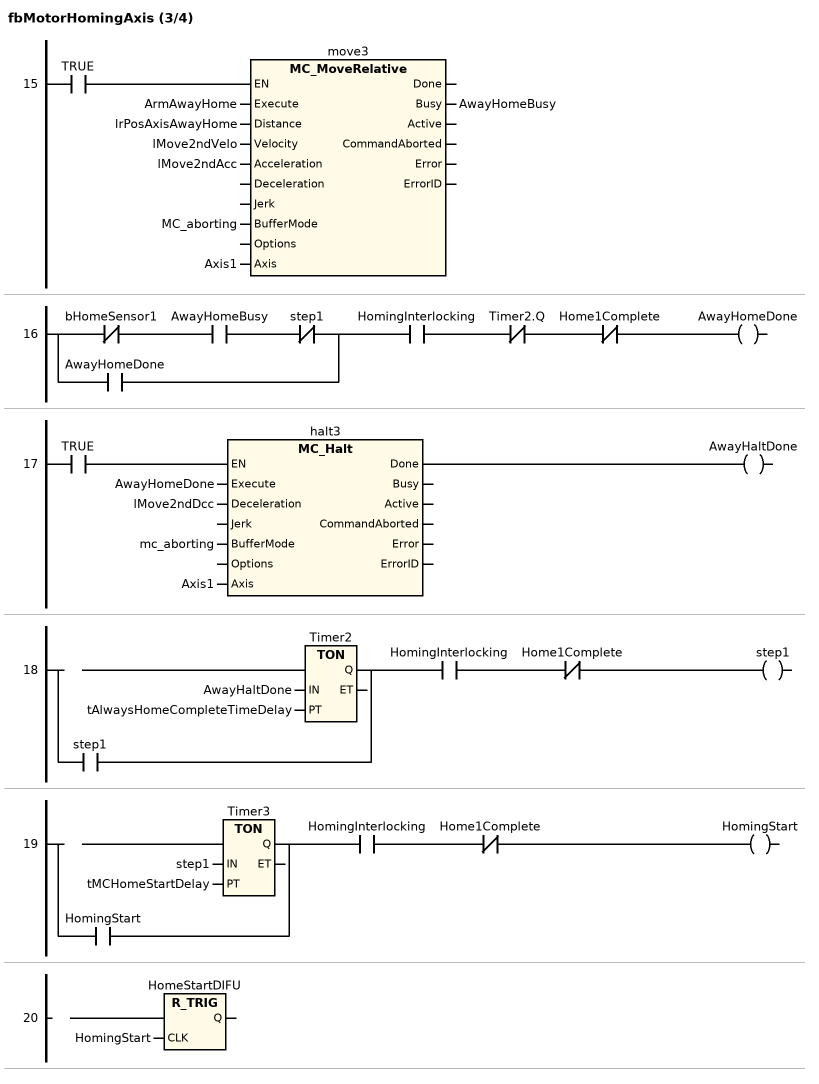
// NETWORK 15
move3(
    Execute := ArmAwayHome,
    Distance := lrPosAxisAwayHome,
    Velocity := lMove2ndVelo,
    Acceleration := lMove2ndAcc,
    BufferMode := MC_aborting,
    Axis := Axis1,
    Busy => AwayHomeBusy); // MC_MoveRelative

// NETWORK 16
AwayHomeDone := (NOT bHomeSensor1 AND AwayHomeBusy AND NOT step1 OR AwayHomeDone) AND HomingInterlocking AND NOT Timer2.Q AND NOT Home1Complete;

// NETWORK 17
halt3(Execute := AwayHomeDone, Deceleration := lMove2ndDcc, BufferMode := mc_aborting, Axis := Axis1); // MC_Halt
AwayHaltDone := halt3.Done;

// NETWORK 18
Timer2(IN := AwayHaltDone, PT := tAlwaysHomeCompleteTimeDelay); // TON
step1 := (Timer2.Q OR step1) AND HomingInterlocking AND NOT Home1Complete;

// NETWORK 19
Timer3(IN := step1, PT := tMCHomeStartDelay); // TON
HomingStart := (Timer3.Q OR HomingStart) AND HomingInterlocking AND NOT Home1Complete;

// NETWORK 20
HomeStartDIFU(CLK := HomingStart); // R_TRIG

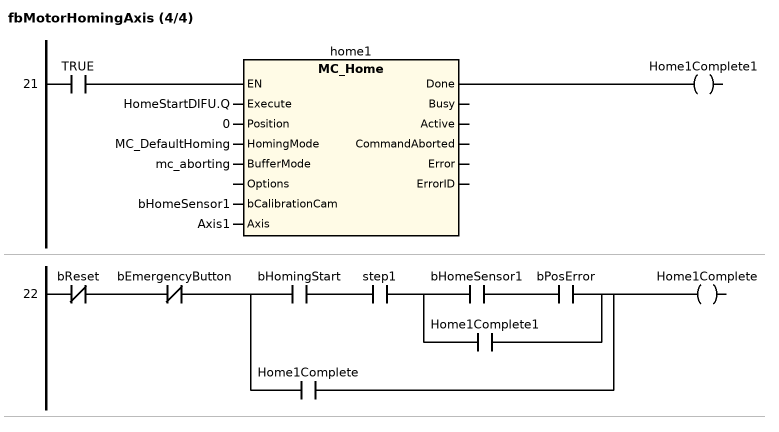
// NETWORK 21
home1(
    Execute := HomeStartDIFU.Q,
    Position := 0,
    HomingMode := MC_DefaultHoming,
    BufferMode := mc_aborting,
    bCalibrationCam := bHomeSensor1,
    Axis := Axis1); // MC_Home
Home1Complete1 := home1.Done;

// NETWORK 22
Home1Complete := NOT bReset AND NOT bEmergencyButton AND (bHomingStart AND step1 AND (bHomeSensor1 AND bPosError OR Home1Complete1) OR Home1Complete);

END_FUNCTION_BLOCK

// ---- FBs/B_JKS_CustomFB/fbArmCtrlFolder/fbMultipleArmAgiCtrl.TcPOU
FUNCTION_BLOCK fbMultipleArmAgiCtrl
VAR_INPUT
	bEN: BOOL;
	bBasketCfm: BOOL;
	bEmergencyStop: BOOL;
	bStnProcessComplete: BOOL;
	bMultiArmAgiDownRS: BOOL;
	bMultiArmAgiMidRS: BOOL;
END_VAR
VAR_OUTPUT
	bMultiArmAgiInProcess: BOOL;
	bMultiArmAgiDown: BOOL;
	bMultiArmAgiUp: BOOL;

END_VAR
VAR

END_VAR

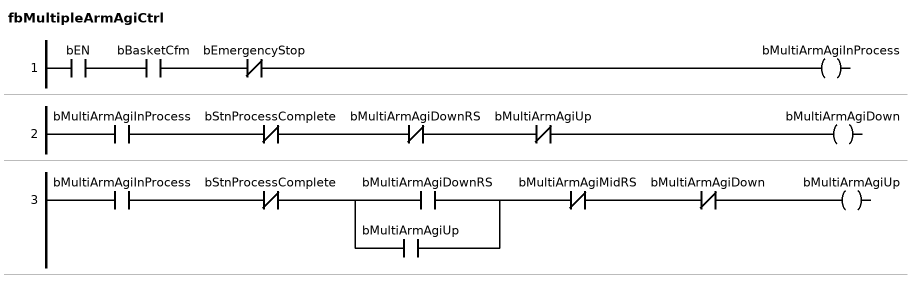
// NETWORK 1
bMultiArmAgiInProcess := bEN AND bBasketCfm AND NOT bEmergencyStop;

// NETWORK 2
bMultiArmAgiDown := bMultiArmAgiInProcess AND NOT bStnProcessComplete AND NOT bMultiArmAgiDownRS AND NOT bMultiArmAgiUp;

// NETWORK 3
bMultiArmAgiUp := (bMultiArmAgiInProcess AND NOT bStnProcessComplete AND (bMultiArmAgiDownRS OR bMultiArmAgiUp)) AND NOT bMultiArmAgiMidRS AND NOT bMultiArmAgiDown;

END_FUNCTION_BLOCK

// ---- FBs/B_JKS_CustomFB/fbArmCtrlFolder/fbSlowPullAxisCtrl.TcPOU
FUNCTION_BLOCK fbSlowPullAxisCtrl
VAR_INPUT

	bPosStart : BOOL;
	bHomingRdy : BOOL;
	wTargetPosNum : WORD;
	lrDownVelo : LREAL;
	lrDownAcc : LREAL;
	lrDownDcc : LREAL;
	lrDownVelo2 : LREAL;
	lrDownAcc2 : LREAL;
	lrDownDcc2 : LREAL;
	lrUpVelo : LREAL;
	lrUpAcc : LREAL;
	lrUpDcc : LREAL;
	lrUpVelo2 : LREAL;
	lrUpAcc2 : LREAL;
	lrUpDcc2: LREAL;
	lrCurrentServoPos : LREAL;
	lrDownPos : LREAL;
	lrUpPos : LREAL;
	lrUpAgitationPos : LREAL;
	lrDownAgitationPos : LREAL;

END_VAR

VAR_IN_OUT

	ArmLifter : axis_ref;
END_VAR

VAR_OUTPUT

	AxisStopEn : BOOL;

END_VAR
VAR

	Halt1: MC_Halt;
	Stoptimer: TON;
	AxisStopbit: BOOL;
	TimerMove: TON;
	BlockStartBit: BOOL;
	Move1: BOOL;
	Move2: BOOL;
	Move3: BOOL;
	Move4: BOOL;
	Move5: BOOL;
	Move6: BOOL;
	Move7: BOOL;
	Move8: BOOL;
	Move9: BOOL;
	Move10: BOOL;
	Move11: BOOL;
	Move12: BOOL;
	Move13: BOOL;
	Move14: BOOL;
	Move15: BOOL;
	Move16: BOOL;
	Move17: BOOL;
	Move18: BOOL;
	Move19: BOOL;
	Move20: BOOL;
	Halt2: MC_Halt;
	ArmMoveTostation2: MC_MoveAbsolute;
	ArmMoveTostation: MC_MoveAbsolute;
	PosSV: LREAL;
	AccSv: LREAL;
	DccSv: LREAL;
	VeloSv: LREAL;
	Arm2ndSpeedEnable: BOOL;

END_VAR
VAR // added by the converter: edge detectors and wires of the graphical bodies
    _w1, _w2, _w3, _w4, _w5, _w6, _w7, _w8, _w9, _w10, _w11, _w12, _w13, _w14, _w15, _w16 : LREAL;
END_VAR

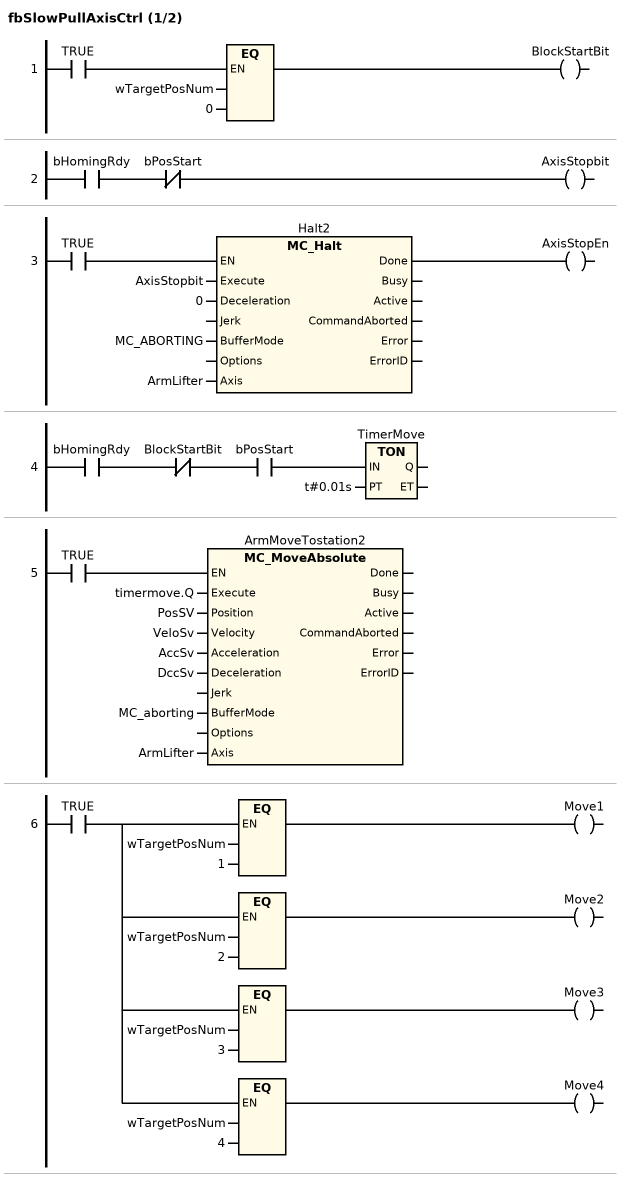
// NETWORK 1
BlockStartBit := wTargetPosNum = 0;

// NETWORK 2
AxisStopbit := bHomingRdy AND NOT bPosStart;

// NETWORK 3
Halt2(Execute := AxisStopbit, Deceleration := 0, BufferMode := MC_ABORTING, Axis := ArmLifter); // MC_Halt
AxisStopEn := Halt2.Done;

// NETWORK 4
TimerMove(IN := bHomingRdy AND NOT BlockStartBit AND bPosStart, PT := t#0.01s); // TON

// NETWORK 5
ArmMoveTostation2(
    Execute := timermove.Q,
    Position := PosSV,
    Velocity := VeloSv,
    Acceleration := AccSv,
    Deceleration := DccSv,
    BufferMode := MC_aborting,
    Axis := ArmLifter); // MC_MoveAbsolute

// NETWORK 6
Move1 := wTargetPosNum = 1;
Move2 := wTargetPosNum = 2;
Move3 := wTargetPosNum = 3;
Move4 := wTargetPosNum = 4;

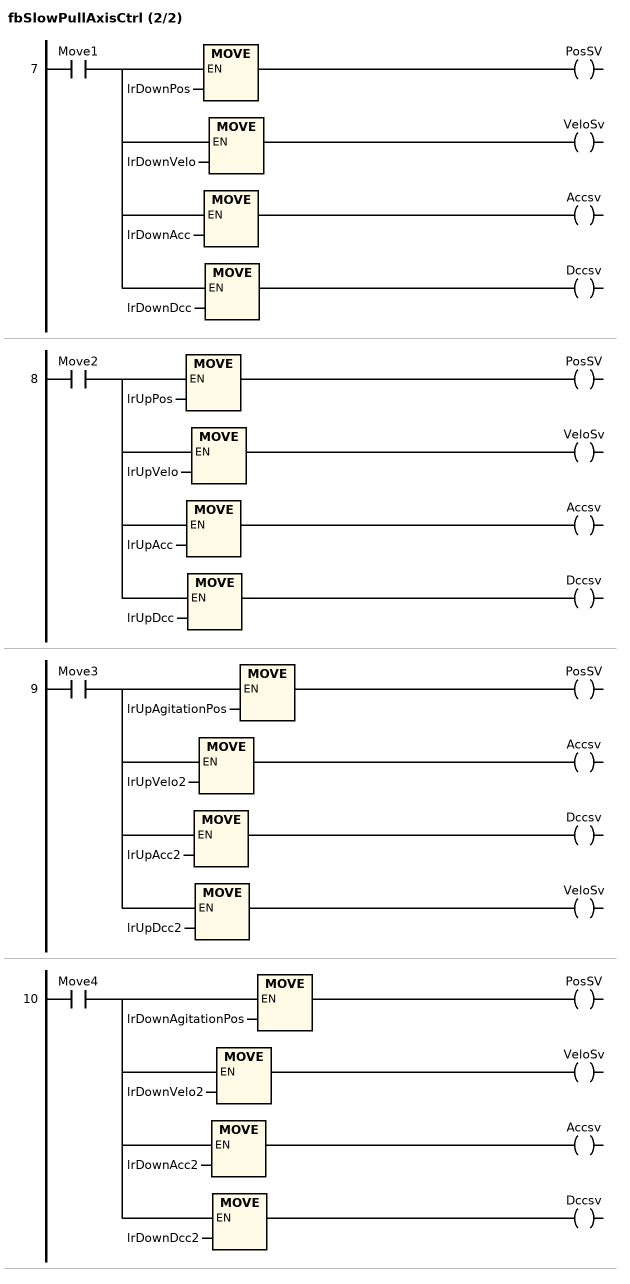
// NETWORK 7
IF Move1 THEN _w1 := lrDownPos; END_IF
PosSV := _w1;
IF Move1 THEN _w2 := lrDownVelo; END_IF
VeloSv := _w2;
IF Move1 THEN _w3 := lrDownAcc; END_IF
Accsv := _w3;
IF Move1 THEN _w4 := lrDownDcc; END_IF
Dccsv := _w4;

// NETWORK 8
IF Move2 THEN _w5 := lrUpPos; END_IF
PosSV := _w5;
IF Move2 THEN _w6 := lrUpVelo; END_IF
VeloSv := _w6;
IF Move2 THEN _w7 := lrUpAcc; END_IF
Accsv := _w7;
IF Move2 THEN _w8 := lrUpDcc; END_IF
Dccsv := _w8;

// NETWORK 9
IF Move3 THEN _w9 := lrUpAgitationPos; END_IF
PosSV := _w9;
IF Move3 THEN _w10 := lrUpVelo2; END_IF
Accsv := _w10;
IF Move3 THEN _w11 := lrUpAcc2; END_IF
Dccsv := _w11;
IF Move3 THEN _w12 := lrUpDcc2; END_IF
VeloSv := _w12;

// NETWORK 10
IF Move4 THEN _w13 := lrDownAgitationPos; END_IF
PosSV := _w13;
IF Move4 THEN _w14 := lrDownVelo2; END_IF
VeloSv := _w14;
IF Move4 THEN _w15 := lrDownAcc2; END_IF
Accsv := _w15;
IF Move4 THEN _w16 := lrDownDcc2; END_IF
Dccsv := _w16;

END_FUNCTION_BLOCK

// ---- FBs/B_JKS_CustomFB/fbArmCtrlFolder/fb_AxisMovement_Down.TcPOU
FUNCTION_BLOCK fb_AxisMovement_Down
VAR_INPUT
	bEstop			: BOOL;
	bHomingReady	: BOOL;
	bMove_Activate	: BOOL;
	DS_Variable		: DS_SA_Movement;
	lrCurrentAxPos	: LREAL;
	wTargerPosNum	: DWORD;
	lrPos1			: LREAL;
	lrPos2			: LREAL;
	lrPos3			: LREAL;
	lrPos4			: LREAL;
	lrPos5			: LREAL;
	lrPos6			: LREAL;
	lrPos7			: LREAL;
	lrPos8			: LREAL;
	lrPos9			: LREAL;
	lrPos10			: LREAL;
	lrPos11			: LREAL;
	lrPos12			: LREAL;
	lrPos13			: LREAL;
	lrPos14			: LREAL;
	lrPos15			: LREAL;
	lrPos16			: LREAL;
	lrPos17			: LREAL;
	lrPos18			: LREAL;
	lrPos19			: LREAL;
	lrPos20			: LREAL;
	iTimeDelay		: TIME;

END_VAR
VAR_IN_OUT
	Ax_1	: Axis_Ref;
	lrPosTolerance	: LREAL;
END_VAR
VAR_OUTPUT
	Ax_MoveComplete	: BOOL;
	Step	: INT;
END_VAR
VAR
	Timer1: BOOL;
	MC_MoveContinuousAbsolute: ARRAY [1..4] OF MC_MoveContinuousAbsolute;
	lrTargetPos: LREAL;
	MC_MoveAbsolute1: MC_MoveAbsolute;
	Timer2: BOOL;

	MC_MoveAbsolute2: MC_MoveAbsolute;
	Timer3: BOOL;

	MC_MoveAbsolute3: MC_MoveAbsolute;
	Timer4: BOOL;

	MC_MoveAbsolute4: MC_MoveAbsolute;
	bHalt: BOOL;
	MC_Stop1: MC_Stop;
	R_TRIG1: R_TRIG;
	R_TRIG2: R_TRIG;
	R_TRIG3: R_TRIG;
	R_TRIG4: R_TRIG;
	bZoneChange : ARRAY [1..4] OF BOOL;



	TON1: TON;
	TON2: TON;
	TON3: TON;
	TON4: TON;
	R_TRIG11: R_TRIG;
	Start: BOOL;
	TON11: TON;
	StartRE: R_TRIG;
	StartFE: F_TRIG;
	bNotHomingReadyRE: R_TRIG;
END_VAR

MC_Stop1(
	Execute:=bHalt ,
	Deceleration:=0 ,
	Jerk:= ,
	Options:= ,
	Axis:=Ax_1 ,
	Done=> ,
	Busy=> ,
	Active=>  );

IF wTargerPosNum = 1 THEN
	lrTargetPos	:= lrPos1;
ELSIF wTargerPosNum = 2 THEN
	lrTargetPos	:= lrPos2;
ELSIF wTargerPosNum = 3 THEN
	lrTargetPos	:= lrPos3;
ELSIF wTargerPosNum = 4 THEN
	lrTargetPos	:= lrPos4;
ELSIF wTargerPosNum = 5 THEN
	lrTargetPos	:= lrPos5;
ELSIF wTargerPosNum = 6 THEN
	lrTargetPos	:= lrPos6;
ELSIF wTargerPosNum = 7 THEN
	lrTargetPos	:= lrPos7;
ELSIF wTargerPosNum = 8 THEN
	lrTargetPos	:= lrPos8;
ELSIF wTargerPosNum = 9 THEN
	lrTargetPos	:= lrPos9;
ELSIF wTargerPosNum = 10 THEN
	lrTargetPos	:= lrPos10;
ELSIF wTargerPosNum = 11 THEN
	lrTargetPos	:= lrPos11;
ELSIF wTargerPosNum = 12 THEN
	lrTargetPos	:= lrPos12;
ELSIF wTargerPosNum = 13 THEN
	lrTargetPos	:= lrPos13;
ELSIF wTargerPosNum = 14 THEN
	lrTargetPos	:= lrPos14;
ELSIF wTargerPosNum = 15 THEN
	lrTargetPos	:= lrPos15;
ELSIF wTargerPosNum = 16 THEN
	lrTargetPos	:= lrPos16;
ELSIF wTargerPosNum = 17 THEN
	lrTargetPos	:= lrPos17;
ELSIF wTargerPosNum = 18 THEN
	lrTargetPos	:= lrPos18;
ELSIF wTargerPosNum = 19 THEN
	lrTargetPos	:= lrPos19;
ELSIF wTargerPosNum = 20 THEN
	lrTargetPos	:= lrPos20;
ELSE
	lrTargetPos	:=0;
END_IF


StartRE(CLK:=Start , Q=> );
StartFE(CLK:=Start , Q=> );
bNotHomingReadyRE(CLK:= NOT bHomingReady , Q=> );

IF bEstop OR bNotHomingReadyRE.Q OR StartFE.Q THEN
	wTargerPosNum	:= 0;
	Step	:= 0;
	bHalt	:= TRUE;
	bZoneChange[1]:=FALSE;
	bZoneChange[2]:=FALSE;
	bZoneChange[3]:=FALSE;
	bZoneChange[4]:=FALSE;
	Ax_MoveComplete	:= FALSE;
ELSE
	bHalt	:= FALSE;
END_IF

IF StartRE.Q THEN
(*Step	:= 0;*)
bZoneChange[1]:=FALSE;
bZoneChange[2]:=FALSE;
bZoneChange[3]:=FALSE;
bZoneChange[4]:=FALSE;
END_IF


IF bHomingReady AND bMove_Activate AND lrTargetPos <> 0  THEN
	Start					:= TRUE;
ELSE
	Start					:= FALSE;
END_IF



R_TRIG1(CLK:=Step=11 , Q=> );
R_TRIG2(CLK:=Step=12 , Q=> );
R_TRIG3(CLK:=Step=13 , Q=> );
R_TRIG4(CLK:=Step=14 , Q=> );

IF lrPosTolerance < 0.1 THEN
lrPosTolerance := 0.1;
ELSIF lrPosTolerance > 5 THEN
lrPosTolerance := 5;
END_IF

IF Start AND NOT bHalt AND NOT  Ax_MoveComplete AND lrCurrentAxPos + lrPosTolerance >=  DS_Variable.lrZone1startPos AND lrCurrentAxPos <  DS_Variable.lrZone2startPos THEN
Step:= 11;
bZoneChange[1]		:=TRUE;
END_IF

IF Start AND NOT bHalt AND NOT Ax_MoveComplete AND lrCurrentAxPos >=  DS_Variable.lrZone2startPos AND lrCurrentAxPos <  DS_Variable.lrZone3startPos THEN
Step:= 12;
bZoneChange[2]		:=TRUE;
END_IF

IF Start AND NOT bHalt AND NOT Ax_MoveComplete AND lrCurrentAxPos >=  DS_Variable.lrZone3startPos AND lrCurrentAxPos <  DS_Variable.lrZone4startPos THEN
Step:= 13;
bZoneChange[3]		:=TRUE;
END_IF

IF Start AND NOT bHalt AND NOT Ax_MoveComplete AND lrCurrentAxPos >=  DS_Variable.lrZone4startPos (*AND lrCurrentAxPos < lrTargetPos*) THEN
Step:= 14;
bZoneChange[4]		:=TRUE;
END_IF

IF Start AND NOT bHalt AND lrCurrentAxPos =  lrTargetPos THEN
Ax_MoveComplete	:= TRUE;
bZoneChange[1]		:=FALSE;
bZoneChange[2]		:=FALSE;
bZoneChange[3]		:=FALSE;
bZoneChange[4]		:=FALSE;
END_IF

CASE Step OF
0:;



11:


		MC_MoveContinuousAbsolute[1](
			Execute:=R_TRIG1.Q(* OR bZoneChange[1] *) ,
			Position:=DS_Variable.lrZone2StartPos ,
			Velocity:=DS_Variable.lrZone1Speed ,
			EndVelocity:=DS_Variable.lrZone2Speed ,
			Acceleration:=DS_Variable.lrZone1Acc ,
			Deceleration:=DS_Variable.lrZone1Dcc ,
			BufferMode:=MC_ABORTING ,
			Axis:=Ax_1 ,
			InEndVelocity=> ,
			Busy=>  );



12:

		MC_MoveContinuousAbsolute[2](
			Execute:=R_TRIG2.Q (*OR bZoneChange[2]*)  ,
			Position:=DS_Variable.lrZone3StartPos ,
			Velocity:=DS_Variable.lrZone2Speed ,
			EndVelocity:=DS_Variable.lrZone3Speed ,
			Acceleration:=DS_Variable.lrZone2Acc ,
			Deceleration:=DS_Variable.lrZone2Dcc ,
			BufferMode:=MC_ABORTING ,
			Axis:=Ax_1 ,
			InEndVelocity=> ,
			Busy=>  );



13:

		MC_MoveContinuousAbsolute[3](
			Execute:=R_TRIG3.Q (*OR bZoneChange[3]*) ,
			Position:=DS_Variable.lrZone4StartPos ,
			Velocity:=DS_Variable.lrZone3Speed ,
			EndVelocity:=DS_Variable.lrZone4Speed ,
			Acceleration:=DS_Variable.lrZone3Acc ,
			Deceleration:=DS_Variable.lrZone3Dcc ,
			BufferMode:=MC_ABORTING ,
			Axis:=Ax_1 ,
			InEndVelocity=> ,
			Busy=>  );

14:

		MC_MoveAbsolute4(
			Execute:=R_TRIG4.Q (*OR bZoneChange[4]*) ,
			Position:=lrTargetPos ,
			Velocity:=DS_Variable.lrZone4Speed ,
			Acceleration:=DS_Variable.lrZone4Acc ,
			Deceleration:=DS_Variable.lrZone4Dcc ,
			BufferMode:=MC_ABORTING ,
			Axis:=Ax_1 ,
			Done=> ,
			Busy=> ,
			Active=>  );
		



END_CASE

END_FUNCTION_BLOCK

// ---- FBs/B_JKS_CustomFB/fbArmCtrlFolder/fb_AxisMovement_Up.TcPOU
FUNCTION_BLOCK fb_AxisMovement_Up
VAR_INPUT
	bEstop			: BOOL;
	bHomingReady	: BOOL;
	bMove_Activate	: BOOL;
	DS_Variable		: DS_SA_Movement;
	lrCurrentAxPos	: LREAL;
	wTargerPosNum	: DWORD;
	lrPos1			: LREAL;
	lrPos2			: LREAL;
	lrPos3			: LREAL;
	lrPos4			: LREAL;
	lrPos5			: LREAL;
	lrPos6			: LREAL;
	lrPos7			: LREAL;
	lrPos8			: LREAL;
	lrPos9			: LREAL;
	lrPos10			: LREAL;
	lrPos11			: LREAL;
	lrPos12			: LREAL;
	lrPos13			: LREAL;
	lrPos14			: LREAL;
	lrPos15			: LREAL;
	lrPos16			: LREAL;
	lrPos17			: LREAL;
	lrPos18			: LREAL;
	lrPos19			: LREAL;
	lrPos20			: LREAL;
	iTimeDelay		: TIME;

END_VAR
VAR_IN_OUT
	Ax_1	: Axis_Ref;
	lrPosTolerance	: LREAL;

END_VAR
VAR_OUTPUT
	Ax_MoveComplete	: BOOL;
	Step	: INT;
END_VAR
VAR
	Timer1: BOOL;
	MC_MoveContinuousAbsolute: ARRAY [1..4] OF MC_MoveContinuousAbsolute;
	lrTargetPos: LREAL;
	MC_MoveAbsolute1: MC_MoveAbsolute;
	Timer2: BOOL;

	MC_MoveAbsolute2: MC_MoveAbsolute;
	Timer3: BOOL;

	MC_MoveAbsolute3: MC_MoveAbsolute;
	Timer4: BOOL;

	MC_MoveAbsolute4: MC_MoveAbsolute;
	bHalt: BOOL;
	MC_Stop1: MC_Stop;
	R_TRIG1: R_TRIG;
	R_TRIG2: R_TRIG;
	R_TRIG3: R_TRIG;
	R_TRIG4: R_TRIG;
	bZoneChange : ARRAY [1..4] OF BOOL;




	TON1: TON;
	TON2: TON;
	TON3: TON;
	TON4: TON;
	R_TRIG11: R_TRIG;
	Start: BOOL;
	TON11: TON;
	StartRE: R_TRIG;
	StartFE: F_TRIG;

	bNotHomingReadyRE: R_TRIG;
END_VAR

MC_Stop1(
	Execute:=bHalt ,
	Deceleration:=0 ,
	Jerk:= ,
	Options:= ,
	Axis:=Ax_1 ,
	Done=> ,
	Busy=> ,
	Active=>  );

IF wTargerPosNum = 1 THEN
	lrTargetPos	:= lrPos1;
ELSIF wTargerPosNum = 2 THEN
	lrTargetPos	:= lrPos2;
ELSIF wTargerPosNum = 3 THEN
	lrTargetPos	:= lrPos3;
ELSIF wTargerPosNum = 4 THEN
	lrTargetPos	:= lrPos4;
ELSIF wTargerPosNum = 5 THEN
	lrTargetPos	:= lrPos5;
ELSIF wTargerPosNum = 6 THEN
	lrTargetPos	:= lrPos6;
ELSIF wTargerPosNum = 7 THEN
	lrTargetPos	:= lrPos7;
ELSIF wTargerPosNum = 8 THEN
	lrTargetPos	:= lrPos8;
ELSIF wTargerPosNum = 9 THEN
	lrTargetPos	:= lrPos9;
ELSIF wTargerPosNum = 10 THEN
	lrTargetPos	:= lrPos10;
ELSIF wTargerPosNum = 11 THEN
	lrTargetPos	:= lrPos11;
ELSIF wTargerPosNum = 12 THEN
	lrTargetPos	:= lrPos12;
ELSIF wTargerPosNum = 13 THEN
	lrTargetPos	:= lrPos13;
ELSIF wTargerPosNum = 14 THEN
	lrTargetPos	:= lrPos14;
ELSIF wTargerPosNum = 15 THEN
	lrTargetPos	:= lrPos15;
ELSIF wTargerPosNum = 16 THEN
	lrTargetPos	:= lrPos16;
ELSIF wTargerPosNum = 17 THEN
	lrTargetPos	:= lrPos17;
ELSIF wTargerPosNum = 18 THEN
	lrTargetPos	:= lrPos18;
ELSIF wTargerPosNum = 19 THEN
	lrTargetPos	:= lrPos19;
ELSIF wTargerPosNum = 20 THEN
	lrTargetPos	:= lrPos20;
ELSE
	lrTargetPos	:=0;
END_IF


StartRE(CLK:=Start , Q=> );
StartFE(CLK:=Start , Q=> );
bNotHomingReadyRE(CLK:= NOT bHomingReady , Q=> );

IF bEstop OR bNotHomingReadyRE.Q OR StartFE.Q THEN
	wTargerPosNum	:= 0;
	Step	:= 0;
	bHalt	:= TRUE;
	bZoneChange[1]:=FALSE;
	bZoneChange[2]:=FALSE;
	bZoneChange[3]:=FALSE;
	bZoneChange[4]:=FALSE;
ELSE
	bHalt	:= FALSE;
END_IF

IF StartRE.Q THEN
Step	:= 0;
bZoneChange[1]:=FALSE;
bZoneChange[2]:=FALSE;
bZoneChange[3]:=FALSE;
bZoneChange[4]:=FALSE;
END_IF


IF bHomingReady AND bMove_Activate AND lrTargetPos <> 0  THEN
	Start					:= TRUE;
ELSE
	Start					:= FALSE;
END_IF


R_TRIG1(CLK:=Step=11 , Q=> );
R_TRIG2(CLK:=Step=12 , Q=> );
R_TRIG3(CLK:=Step=13 , Q=> );
R_TRIG4(CLK:=Step=14 , Q=> );

IF lrPosTolerance < 0.1 THEN
lrPosTolerance := 0.1;
ELSIF lrPosTolerance > 5 THEN
lrPosTolerance := 5;
END_IF

IF Start AND NOT bHalt AND NOT  Ax_MoveComplete AND lrCurrentAxPos - lrPosTolerance <=  DS_Variable.lrZone1startPos AND lrCurrentAxPos >  DS_Variable.lrZone2startPos THEN
Step:= 11;
bZoneChange[1]		:=TRUE;
END_IF

IF Start AND NOT bHalt AND NOT Ax_MoveComplete AND lrCurrentAxPos <=  DS_Variable.lrZone2startPos AND lrCurrentAxPos >  DS_Variable.lrZone3startPos THEN
Step:= 12;
bZoneChange[2]		:=TRUE;
END_IF

IF Start AND NOT bHalt AND NOT Ax_MoveComplete AND lrCurrentAxPos <=  DS_Variable.lrZone3startPos AND lrCurrentAxPos >  DS_Variable.lrZone4startPos THEN
Step:= 13;
bZoneChange[3]		:=TRUE;
END_IF

IF Start AND NOT bHalt AND NOT Ax_MoveComplete AND lrCurrentAxPos <=  DS_Variable.lrZone4startPos (*AND lrCurrentAxPos > lrTargetPos*) THEN
Step:= 14;
bZoneChange[4]		:=TRUE;
END_IF

IF Start AND NOT bHalt AND lrCurrentAxPos =  lrTargetPos THEN
Ax_MoveComplete	:= TRUE;
bZoneChange[1]		:=FALSE;
bZoneChange[2]		:=FALSE;
bZoneChange[3]		:=FALSE;
bZoneChange[4]		:=FALSE;
END_IF

CASE Step OF
0:;



11:



		MC_MoveContinuousAbsolute[1](
			Execute:=R_TRIG1.Q (*OR bZoneChange[1]*)  ,
			Position:=DS_Variable.lrZone2StartPos ,
			Velocity:=DS_Variable.lrZone1Speed ,
			EndVelocity:=DS_Variable.lrZone2Speed ,
			Acceleration:=DS_Variable.lrZone1Acc ,
			Deceleration:=DS_Variable.lrZone1Dcc ,
			BufferMode:=MC_ABORTING ,
			Axis:=Ax_1 ,
			InEndVelocity=> ,
			Busy=>  );



12:

		MC_MoveContinuousAbsolute[2](
			Execute:=R_TRIG2.Q (*OR bZoneChange[2]*)  ,
			Position:=DS_Variable.lrZone3StartPos ,
			Velocity:=DS_Variable.lrZone2Speed ,
			EndVelocity:=DS_Variable.lrZone3Speed ,
			Acceleration:=DS_Variable.lrZone2Acc ,
			Deceleration:=DS_Variable.lrZone2Dcc ,
			BufferMode:=MC_ABORTING ,
			Axis:=Ax_1 ,
			InEndVelocity=> ,
			Busy=>  );



13:


		MC_MoveContinuousAbsolute[3](
			Execute:=R_TRIG3.Q (*OR bZoneChange[3]*) ,
			Position:=DS_Variable.lrZone4StartPos ,
			Velocity:=DS_Variable.lrZone3Speed ,
			EndVelocity:=DS_Variable.lrZone4Speed ,
			Acceleration:=DS_Variable.lrZone3Acc ,
			Deceleration:=DS_Variable.lrZone3Dcc ,
			BufferMode:=MC_ABORTING ,
			Axis:=Ax_1 ,
			InEndVelocity=> ,
			Busy=>  );

14:


		MC_MoveAbsolute4(
			Execute:=R_TRIG4.Q (*OR bZoneChange[4]*) ,
			Position:=lrTargetPos ,
			Velocity:=DS_Variable.lrZone4Speed ,
			Acceleration:=DS_Variable.lrZone4Acc ,
			Deceleration:=DS_Variable.lrZone4Dcc ,
			BufferMode:=MC_ABORTING ,
			Axis:=Ax_1 ,
			Done=> ,
			Busy=> ,
			Active=>  );
		



END_CASE

END_FUNCTION_BLOCK

// ---- FBs/B_JKS_CustomFB/fbArmCtrlFolder/FB_DRIVE_STATUS_ONE_AX.TcPOU
FUNCTION_BLOCK FB_DRIVE_STATUS_ONE_AX
VAR_INPUT

END_VAR
VAR_OUTPUT
	DrvDiag_Err:BOOL;
	DrvRst_Bs:BOOL;
	DrvRst_Err:BOOL;
	fbRdClsXDiag_Ax1_ClsXDiag  	: WORD;

	stC1D_Ax1  : ST_AX5000_C1D;

	AxsErr_Ax1:BOOL;

	AxsSts_Ax1:ST_AxisStatus;

END_VAR
VAR
	fbRdClsXDiag_Ax1:FB_SoEReadClassXDiag;
	fbRdClsXDiag_Ax1_Ex: BOOL;
	fbRdClsXDiag_Ax1_Bs 		: BOOL;
	fbRdClsXDiag_Ax1_Err 		: BOOL;
	fbRdClsXDiag_Ax1_AdsErrId 		: UINT;
	fbRdClsXDiag_Ax1_SerErrId 	: UINT;

	fbRdClsXDiag_Ax1_Att 	: DWORD;


	fbSOERst_Ax1:FB_SoEReset;
	fbSOERst_Ax1_Ex:BOOL;
	fbSOERst_Ax1_Bs 		: BOOL;
	fbSOERst_Ax1_Err 		: BOOL;
	fbSOERst_Ax1_AdsErrId 		: UINT;
	fbSOERst_Ax1_SerErrId 	: UINT;


	fbAxRst_Ax1:MC_Reset;


	step: INT;
	DiagTrig:R_TRIG;
	RstTrig:R_TRIG;
END_VAR

VAR_IN_OUT
	AX_1:Axis_Ref;
	DrvDiag_Ex:BOOL;
	DrvRst_Ex:BOOL;
END_VAR

AX_1.ReadStatus();


AxsSts_Ax1:=AX_1.Status;


AxsErr_Ax1:= AX_1.Status.Error;

RstTrig(CLK:=DrvRst_Ex, Q=> );
IF RstTrig.Q THEN
step:=10;
	DrvRst_Bs:=FALSE;
	DrvRst_Err:=FALSE;
END_IF

DiagTrig(CLK:=DrvDiag_Ex, Q=> );
IF DiagTrig.Q THEN
	step:=1;
END_IF



CASE step OF
	0: (*do nothing*)
	step:=1;

	1:
	fbRdClsXDiag_Ax1(
	NetId:='' ,
	Execute:=TRUE ,
	DiagClass:=1 ,
	Timeout:=DEFAULT_ADS_TIMEOUT ,
	Axis:=AX_1 ,
	Busy=> fbRdClsXDiag_Ax1_Bs,
	Error=> fbRdClsXDiag_Ax1_Err,
	AdsErrId=>fbRdClsXDiag_Ax1_AdsErrId,
	SercosErrId=>fbRdClsXDiag_Ax1_SerErrId ,
	ClassXDiag=>fbRdClsXDiag_Ax1_ClsXDiag ,
	Attribute=> fbRdClsXDiag_Ax1_Att);
	stC1D_Ax1:=F_ConvWordToSTAX5000C1D(fbRdClsXDiag_Ax1_ClsXDiag);
	step:=2;

	2:
	fbRdClsXDiag_Ax1(
	NetId:='' ,
	Execute:=TRUE ,
	DiagClass:=1 ,
	Timeout:=DEFAULT_ADS_TIMEOUT ,
	Axis:=AX_1 ,
	Busy=> fbRdClsXDiag_Ax1_Bs,
	Error=> fbRdClsXDiag_Ax1_Err,
	AdsErrId=>fbRdClsXDiag_Ax1_AdsErrId,
	SercosErrId=>fbRdClsXDiag_Ax1_SerErrId ,
	ClassXDiag=>fbRdClsXDiag_Ax1_ClsXDiag ,
	Attribute=> fbRdClsXDiag_Ax1_Att);
	stC1D_Ax1:=F_ConvWordToSTAX5000C1D(fbRdClsXDiag_Ax1_ClsXDiag);
	IF NOT fbRdClsXDiag_Ax1_Bs THEN
	step:=3;
	END_IF

	3:
	fbRdClsXDiag_Ax1(
	NetId:='' ,
	Execute:=FALSE ,
	DiagClass:=1 ,
	Timeout:=DEFAULT_ADS_TIMEOUT ,
	Axis:=AX_1 ,
	Busy=> fbRdClsXDiag_Ax1_Bs,
	Error=> fbRdClsXDiag_Ax1_Err,
	AdsErrId=>fbRdClsXDiag_Ax1_AdsErrId,
	SercosErrId=>fbRdClsXDiag_Ax1_SerErrId ,
	ClassXDiag=>fbRdClsXDiag_Ax1_ClsXDiag ,
	Attribute=> fbRdClsXDiag_Ax1_Att);
	stC1D_Ax1:=F_ConvWordToSTAX5000C1D(fbRdClsXDiag_Ax1_ClsXDiag);
	step:=4;

	4:
	DrvDiag_Ex:=FALSE;
	IF  fbRdClsXDiag_Ax1_ClsXDiag <> 0 THEN
		DrvDiag_Err:=TRUE;
	ELSE
		DrvDiag_Err:=FALSE;
	END_IF
	step:=1;

	10:
	DrvRst_Bs:=TRUE;
	step:=11;

	11:
	fbSOERst_Ax1(
	NetId:= ,
	Execute:=TRUE ,
	Timeout:=DEFAULT_ADS_TIMEOUT ,
	Axis:=AX_1 ,
	Busy=>fbSOERst_Ax1_Bs ,
	Error=>fbSOERst_Ax1_Err ,
	AdsErrId=>fbSOERst_Ax1_AdsErrId ,
	SercosErrId=> fbSOERst_Ax1_SerErrId);
	step:=12;

	12:
	fbSOERst_Ax1(
	NetId:= ,
	Execute:=TRUE ,
	Timeout:=DEFAULT_ADS_TIMEOUT ,
	Axis:=AX_1 ,
	Busy=>fbSOERst_Ax1_Bs ,
	Error=>fbSOERst_Ax1_Err ,
	AdsErrId=>fbSOERst_Ax1_AdsErrId ,
	SercosErrId=> fbSOERst_Ax1_SerErrId);
	IF NOT fbSOERst_Ax1_Bs THEN
	step:=13;
	END_IF

	13:
	fbSOERst_Ax1(
	NetId:= ,
	Execute:=FALSE ,
	Timeout:=DEFAULT_ADS_TIMEOUT ,
	Axis:=AX_1 ,
	Busy=>fbSOERst_Ax1_Bs ,
	Error=>fbSOERst_Ax1_Err ,
	AdsErrId=>fbSOERst_Ax1_AdsErrId ,
	SercosErrId=> fbSOERst_Ax1_SerErrId);
	step:=17;

	17:
	fbAxRst_Ax1(
	Execute:=TRUE ,
	Axis:=Ax_1 ,
	Done=> ,
	Busy=> , 
	Error=> , 
	ErrorID=> );
	step:=18;

	18:
	fbAxRst_Ax1(
	Execute:=TRUE ,
	Axis:=Ax_1 ,
	Done=> ,
	Busy=> , 
	Error=> , 
	ErrorID=> );
	IF NOT fbAxRst_Ax1.Busy THEN
		step:=19;
	END_IF

	19:
	fbAxRst_Ax1(
	Execute:=FALSE ,
	Axis:=Ax_1 ,
	Done=> ,
	Busy=> ,
	Error=> ,
	ErrorID=> );
	step:=23;

	23:
	DrvRst_Bs:=FALSE;
	DrvRst_Ex:=FALSE;
	step:=1;

END_CASE

END_FUNCTION_BLOCK

// ---- FBs/B_JKS_CustomFB/fbBarcodeCtrl/fbBarcodeScanner.TcPOU
FUNCTION_BLOCK fbBarcodeScanner
VAR_INPUT

	bON							: BOOL;

END_VAR

VAR_OUTPUT

	sSendString						: STRING;
	sReceivedString					: STRING;

END_VAR

VAR_IN_OUT

	cbComBufferWrite 					: ComBuffer;
	cbComBufferRead 				: ComBuffer;


END_VAR

VAR
	bEnable  						: BOOL := TRUE;
	bSendString						: BOOL;
	fbTON_1s						: TON;
	bON_Delay						: TON;
	bOFF_Reflash					: TON;

	R_TRIG_ON						: R_TRIG;
	R_TRIG_OFF						: R_TRIG;


	step								:BYTE;

	fbReceiveString 					: ReceiveString;
	fbReceiveString_Rst				: BOOL;
	fbReceiveString_StrRcv			: BOOL;

	fbSendString255					: SendString;
	busy							: BOOL;
	error							: comerror_t;

	DelimiteChar						:STRING:='$R';
	sReceivedStringRaw				: STRING;
	iReceivedStingProcess			: INT;

	sReceivedStringRaw2: STRING;
END_VAR

(*bON is "ON" --> Trigger 1 time sending*)

bON_Delay(IN:=bON, PT:=t#0.5s , Q=> , ET=> );

R_TRIG_ON(CLK:=bON_Delay.Q AND bON,Q=>);
IF R_TRIG_ON.Q THEN
	step:= 10;
END_IF

(*bON is "OFF" --> Trigger always OFF reflash*)

bOFF_Reflash(IN:=NOT bOFF_Reflash.Q AND NOT bON, PT:=t#1s , Q=> , ET=> );

R_TRIG_OFF(CLK:=bOFF_Reflash.Q AND NOT bON,Q=>);
IF R_TRIG_OFF.Q THEN
	step:= 20;
END_IF


IF bEnable THEN
	CASE step OF
	0:;

	10:
	sSendString:=CONCAT('LON','$R'); (*ON*)
	step:=0;

	20:
	sSendString:=CONCAT('LOFF','$R'); (*OFF*)
	step:=0;

END_CASE

END_IF

fbReceiveString(
	Prefix:='' ,
	Suffix:='$R',
	Timeout:=t#1s ,
	Reset:=fbReceiveString_Rst ,
	ReceivedString:=sReceivedStringRaw ,
	RXbuffer:=cbComBufferRead ,
	StringReceived=>fbReceiveString_StrRcv ,
	Busy=> ,
	Error=> ,
	RxTimeout=> );

fbTON_1s(IN:=NOT  fbTON_1s.Q, PT:=t#1s , Q=> , ET=> );
bSendString:=fbTON_1s.Q;

IF bSendString AND NOT fbSendString255.Busy THEN
fbSendString255(
	SendString:=sSendString ,
	TXbuffer:=cbComBufferWrite,
	Busy=>busy ,
	Error=> error);
END_IF

IF bON THEN
(*this will find where is the $R located in the string*)
iReceivedStingProcess:=FIND(sReceivedStringRaw, DelimiteChar);

(*after you know the location, you can move the string to another string according to the size*)
sReceivedStringRaw2:=LEFT(sReceivedStringRaw, iReceivedStingProcess-1);

ELSE

sReceivedString := '';
sReceivedStringRaw := 'ERROR$R';

END_IF

IF sReceivedStringRaw2 <> 'ERROR' AND bON THEN

sReceivedString := sReceivedStringRaw2;

ELSE

sReceivedString := '';

END_IF

END_FUNCTION_BLOCK

// ---- FBs/B_JKS_CustomFB/fbBarcodeCtrl/fbBarcodeTrancerNoCode.TcPOU
FUNCTION_BLOCK fbBarcodeTrancerNoCode
VAR_INPUT
	bTracerST : BOOL;
	iTargetProgramNo : INT;
	AR99sProgramNo : ARRAY [0..99] OF STRING;
	AR99sBarcodeDescrip	: ARRAY [0..99] OF STRING;


END_VAR
VAR_OUTPUT

	bProTraceSuccess : BOOL;
	bProTraceFail 	: BOOL;
	iProInRecipeNo 	: INT;
	sProInDescrip	: STRING;
	sProBarCode		: STRING;
END_VAR
VAR
	i: INT;
	TracerRE : R_TRIG;

END_VAR

TracerRE(CLK:=bTracerST,Q=>);

IF NOT bTracerST THEN
	bProTraceSuccess := FALSE;
	bProTraceFail := FALSE;
	iProInRecipeNo := 0;
	i := 1;
END_IF

IF bTracerST AND iTargetProgramNo <> 0 THEN
		FOR i := 1 TO 99 DO

		IF iTargetProgramNo = i THEN
		sProInDescrip := AR99sBarcodeDescrip[i];
		sProBarCode := AR99sProgramNo[i];
		iProInRecipeNo := i;
		bProTraceSuccess := TRUE;
		i := 100;
		END_IF

		END_FOR

END_IF
IF (i > 99 AND bTracerST AND NOT bProTraceSuccess) (*OR (sTargetBarcode = '')*) THEN
bProTraceFail := TRUE;
END_IF

END_FUNCTION_BLOCK

// ---- FBs/B_JKS_CustomFB/fbConversionCtrl/fbRawRatioConversionAllenINV.TcPOU
FUNCTION_BLOCK fbRawRatioConversionAllenINV
VAR_INPUT

	iRawData : INT;
	rRawRatio : LREAL;


END_VAR
VAR_OUTPUT

	rConvertedResult : INT;
END_VAR
VAR
	rRawData: LREAL;
	rConvertedResult_1: LREAL;
END_VAR

rRawData := INT_TO_LREAL (iRawData);

IF rRawData <> 0 AND rRawRatio <> 0 THEN
rConvertedResult_1 := rRawData * rRawRatio;
END_IF

IF rRawData = 0 OR rRawRatio = 0 THEN
rConvertedResult := 0;
END_IF

rConvertedResult := LREAL_TO_INT(rConvertedResult_1);

END_FUNCTION_BLOCK

// ---- FBs/B_JKS_CustomFB/fbConversionCtrl/fbRawRatioConversionUs.TcPOU
FUNCTION_BLOCK fbRawRatioConversionUs
VAR_INPUT

	iRawData : INT;
	rRawRatio : LREAL;


END_VAR
VAR_OUTPUT

	rConvertedResult : INT;
END_VAR
VAR
	rRawData: LREAL;
	rConvertedResult_1: LREAL;
END_VAR

rRawData := INT_TO_LREAL (iRawData);

IF rRawData <> 0 AND rRawRatio <> 0 THEN
rConvertedResult_1 := rRawData * rRawRatio;
END_IF

IF rRawData = 0 OR rRawRatio = 0 THEN
rConvertedResult := 0;
END_IF

rConvertedResult := LREAL_TO_INT(rConvertedResult_1);

END_FUNCTION_BLOCK

// ---- FBs/B_JKS_CustomFB/fbConversionCtrl/fbRawRatioConversionUsPercent.TcPOU
FUNCTION_BLOCK fbRawRatioConversionUsPercent
VAR_INPUT
	iUsRawDataFeedback_Watt 					: INT;
	iUsRawDataOutput_Percent 					: INT;
	lrUsRawRatio_Percent 							: LREAL;
	lrUsMaxData_Watt							: LREAL;
	iUsRawDataOutput_PercentTolerance			: INT;
	tUsRawDataFeedback_PercentCfmDelayOnTime 	: TIME;
	bOutputUs									: BOOL;
END_VAR

VAR_OUTPUT
	iUsFeedbackConvertedResult_Percent			: INT;
	iUsOutputConvertedResult_Watt					: INT;
	bUsFeedbackInRange							: BOOL;
END_VAR

VAR
	lrUsRawDataFeedback_Watt					: LREAL;
	lrUsRawDataOutput_Percent 					: LREAL;
	lrUsFeedbackConvertedResult_Percent			: LREAL;
	lrUsOutputConvertedResult_Watt				: LREAL;
	iUsPercentToleranceP							: INT;
	iUsPercentToleranceN							: INT;
END_VAR

VAR PERSISTENT
	tDelayTimer 									: TON;
END_VAR

(*Converted the US feedback of UsRawDataFeedback_Watt into UsRawDataFeedback_percent *)
lrUsRawDataFeedback_Watt := INT_TO_LREAL (iUsRawDataFeedback_Watt);

IF lrUsRawDataFeedback_Watt <> 0 AND lrUsRawRatio_Percent <> 0 AND lrUsMaxData_Watt <> 0 THEN
lrUsFeedbackConvertedResult_percent := (lrUsRawDataFeedback_Watt / lrUsMaxData_Watt) * lrUsRawRatio_Percent;
END_IF

IF lrUsRawDataFeedback_Watt = 0 OR lrUsRawRatio_Percent = 0 THEN
lrUsFeedbackConvertedResult_percent := 0;
END_IF

iUsFeedbackConvertedResult_percent := LREAL_TO_INT(lrUsFeedbackConvertedResult_percent);

(*Converted the US Output of UsRawDataOutput_Percent into UsRawDataOutput_Watt *)
lrUsRawDataOutput_Percent := INT_TO_LREAL (iUsRawDataOutput_Percent);

IF lrUsRawDataOutput_Percent <> 0 AND lrUsRawRatio_Percent <> 0 AND lrUsMaxData_Watt <> 0 THEN
lrUsOutputConvertedResult_Watt := (lrUsRawDataOutput_Percent / lrUsRawRatio_Percent) * lrUsMaxData_Watt;
END_IF

IF lrUsRawDataOutput_Percent = 0 OR lrUsRawRatio_Percent = 0 THEN
lrUsOutputConvertedResult_Watt := 0;
END_IF

iUsOutputConvertedResult_Watt := LREAL_TO_INT(lrUsOutputConvertedResult_Watt);

(*Fix the tolerance to control US Feedack in Range *)
IF bOutputUS THEN
iUsPercentToleranceP := iUsRawDataOutput_Percent + iUsRawDataOutput_PercentTolerance;
iUsPercentToleranceN := iUsRawDataOutput_Percent - iUsRawDataOutput_PercentTolerance;
END_IF

IF bOutputUS THEN

	tDelayTimer(IN:= iUsFeedbackConvertedResult_Percent >= iUsPercentToleranceN AND iUsFeedbackConvertedResult_Percent <= iUsPercentToleranceP , PT:= tUsRawDataFeedback_PercentCfmDelayOnTime, Q=> , ET=> );

	IF tDelayTimer.Q THEN
	bUSfeedbackInRange := TRUE;
	ELSE
	bUSfeedbackInRange := FALSE;
	END_IF

ELSIF NOT bOutputUS THEN

	bUSfeedbackInRange := FALSE;

ELSE
	bUSfeedbackInRange := FALSE;
END_IF

END_FUNCTION_BLOCK

// ---- FBs/B_JKS_CustomFB/fbDataLogCtrl/F_jx_TS_TO_DATE_STRING.TcPOU
FUNCTION F_jx_TS_TO_DATE_STRING : STRING
VAR_INPUT
	ts_TimeNow: TIMESTRUCT;
	sSeperator: STRING := '/';
END_VAR
VAR
	sDate: STRING;
END_VAR

sDate:='';
sDate:=CONCAT(sDate,WORD_TO_STRING(ts_TimeNow.wDay));
sDate:=CONCAT(sDate,sSeperator);
sDate:=CONCAT(sDate,WORD_TO_STRING(ts_TimeNow.wMonth));
sDate:=CONCAT(sDate,sSeperator);
sDate:=CONCAT(sDate,WORD_TO_STRING(ts_TimeNow.wYear));
F_jx_TS_TO_DATE_STRING:=sDate;

END_FUNCTION

// ---- FBs/B_JKS_CustomFB/fbGeneralfbFolder/UserlevelFB.TcPOU
FUNCTION_BLOCK UserlevelFB
VAR_INPUT
	fb_userlogin:STRING;
	fb_userpassword:ARRAY [0..7] OF STRING;
	fb_username:ARRAY [0..7] OF WSTRING;
END_VAR
VAR_OUTPUT
	fb_userlevel:DWORD;
	fb_userlevelname:WSTRING;
	fb_userloginrecord:ARRAY [0..7] OF BOOL;
END_VAR
VAR
	n: INT;
END_VAR

IF fb_userlogin = fb_userpassword[1] THEN
fb_userlevelname:=fb_username[1];
fb_userlevel:=1;
fb_userloginrecord[0]:=FALSE;
fb_userloginrecord[1]:=TRUE;
fb_userloginrecord[2]:=FALSE;
fb_userloginrecord[3]:=FALSE;
fb_userloginrecord[4]:=FALSE;
fb_userloginrecord[5]:=FALSE;
fb_userloginrecord[6]:=FALSE;
fb_userloginrecord[7]:=FALSE;

ELSIF fb_userlogin = fb_userpassword[2] THEN
fb_userlevel:=2;
fb_userlevelname:=fb_username[2];
fb_userloginrecord[0]:=FALSE;
fb_userloginrecord[1]:=FALSE;
fb_userloginrecord[2]:=TRUE;
fb_userloginrecord[3]:=FALSE;
fb_userloginrecord[4]:=FALSE;
fb_userloginrecord[5]:=FALSE;
fb_userloginrecord[6]:=FALSE;
fb_userloginrecord[7]:=FALSE;

ELSIF fb_userlogin = fb_userpassword[3] THEN
fb_userlevel:=3;
fb_userlevelname:=fb_username[3];
fb_userloginrecord[0]:=FALSE;
fb_userloginrecord[1]:=FALSE;
fb_userloginrecord[2]:=FALSE;
fb_userloginrecord[3]:=TRUE;
fb_userloginrecord[4]:=FALSE;
fb_userloginrecord[5]:=FALSE;
fb_userloginrecord[6]:=FALSE;
fb_userloginrecord[7]:=FALSE;

ELSIF fb_userlogin = fb_userpassword[4] THEN
fb_userlevel:=4;
fb_userlevelname:=fb_username[4];
fb_userloginrecord[0]:=FALSE;
fb_userloginrecord[1]:=FALSE;
fb_userloginrecord[2]:=FALSE;
fb_userloginrecord[3]:=FALSE;
fb_userloginrecord[4]:=TRUE;
fb_userloginrecord[5]:=FALSE;
fb_userloginrecord[6]:=FALSE;
fb_userloginrecord[7]:=FALSE;

ELSIF fb_userlogin = fb_userpassword[5] THEN
fb_userlevel:=5;
fb_userlevelname:=fb_username[5];
fb_userloginrecord[0]:=FALSE;
fb_userloginrecord[1]:=FALSE;
fb_userloginrecord[2]:=FALSE;
fb_userloginrecord[3]:=FALSE;
fb_userloginrecord[4]:=FALSE;
fb_userloginrecord[5]:=TRUE;
fb_userloginrecord[6]:=FALSE;
fb_userloginrecord[7]:=FALSE;

ELSIF fb_userlogin = fb_userpassword[6] THEN
fb_userlevel:=6;
fb_userlevelname:=fb_username[6];
fb_userloginrecord[0]:=FALSE;
fb_userloginrecord[1]:=FALSE;
fb_userloginrecord[2]:=FALSE;
fb_userloginrecord[3]:=FALSE;
fb_userloginrecord[4]:=FALSE;
fb_userloginrecord[5]:=FALSE;
fb_userloginrecord[6]:=TRUE;
fb_userloginrecord[7]:=FALSE;

ELSIF fb_userlogin = fb_userpassword[7] THEN
fb_userlevel:=7;
fb_userlevelname:=fb_username[7];
fb_userloginrecord[0]:=FALSE;
fb_userloginrecord[1]:=FALSE;
fb_userloginrecord[2]:=FALSE;
fb_userloginrecord[3]:=FALSE;
fb_userloginrecord[4]:=FALSE;
fb_userloginrecord[5]:=FALSE;
fb_userloginrecord[6]:=FALSE;
fb_userloginrecord[7]:=TRUE;

ELSE
fb_userlevel:=0;
fb_userlevelname:=fb_username[0];
fb_userloginrecord[0]:=TRUE;
fb_userloginrecord[1]:=FALSE;
fb_userloginrecord[2]:=FALSE;
fb_userloginrecord[3]:=FALSE;
fb_userloginrecord[4]:=FALSE;
fb_userloginrecord[5]:=FALSE;
fb_userloginrecord[6]:=FALSE;
fb_userloginrecord[7]:=FALSE;
END_IF

END_FUNCTION_BLOCK

// ---- FBs/B_JKS_CustomFB/fbStnDegassingCtrl/fbStnDegassCtrl.TcPOU
FUNCTION_BLOCK fbStnDegassCtrl
VAR_INPUT

	bEN								: BOOL;
	bEmergencyStop					: BOOL;
	bVacPumpDeact					: BOOL;
	bDegassPumpDeact				: BOOL;
	bCCHighVacuumSignal			: BOOL;
	bDCHighVacuumSignal			: BOOL;
	bDCLowVacuumSignal				: BOOL;

END_VAR

VAR_OUTPUT
	bDegassInProcess				: BOOL;
	bVacPumpOnOff					: BOOL;
	bDegassPumpOnOff				: BOOL;
(*	bCCVacSuctionValveOnOff			: BOOL;*)
	bDCAirReleaseValveOnOff			: BOOL;
	bDCValveOnOff					: BOOL;
END_VAR

VAR

	bStep1							: BOOL;
	bStep2							: BOOL;
	bStep3							: BOOL;

	TON1							: TON;
	TON2							: TON;
	TON3							: TON;

END_VAR
VAR // added by the converter: edge detectors and wires of the graphical bodies
    _w1 : BOOL;
END_VAR

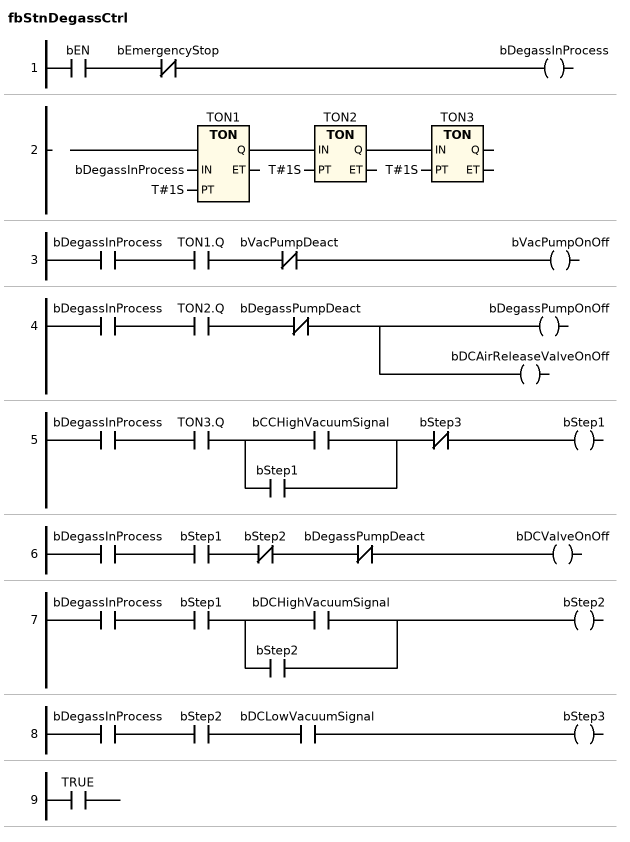
// NETWORK 1
bDegassInProcess := bEN AND NOT bEmergencyStop;

// NETWORK 2
TON1(IN := bDegassInProcess, PT := T#1S); // TON
TON2(IN := TON1.Q, PT := T#1S); // TON
TON3(IN := TON2.Q, PT := T#1S); // TON

// NETWORK 3
bVacPumpOnOff := bDegassInProcess AND TON1.Q AND NOT bVacPumpDeact;

// NETWORK 4
_w1 := bDegassInProcess AND TON2.Q AND NOT bDegassPumpDeact;
bDegassPumpOnOff := _w1;
bDCAirReleaseValveOnOff := _w1;

// NETWORK 5
bStep1 := (bDegassInProcess AND TON3.Q AND (bCCHighVacuumSignal OR bStep1)) AND NOT bStep3;

// NETWORK 6
bDCValveOnOff := bDegassInProcess AND bStep1 AND NOT bStep2 AND NOT bDegassPumpDeact;

// NETWORK 7
bStep2 := bDegassInProcess AND bStep1 AND (bDCHighVacuumSignal OR bStep2);

// NETWORK 8
bStep3 := bDegassInProcess AND bStep2 AND bDCLowVacuumSignal;

// NETWORK 9

END_FUNCTION_BLOCK

// ---- FBs/B_JKS_CustomFB/fbUltrasonicCtrl/BrensonFreqSelector.TcPOU
FUNCTION_BLOCK BrensonFreqSelector
VAR_INPUT
	bSwitch : BOOL;

END_VAR
VAR_IN_OUT

	iFreqAdd : INT;


END_VAR
VAR
	SwitchDF: R_TRIG;
	step : BYTE;

END_VAR

SwitchDF (CLK:=bSwitch , Q=> );

IF iFreqAdd <> 40 AND iFreqAdd <> 80 AND iFreqAdd <> 120 THEN
iFreqAdd := 40;
END_IF

IF SwitchDF.Q AND iFreqAdd = 40 THEN
step := 1;
END_IF

IF SwitchDF.Q AND iFreqAdd = 80 THEN
step := 2;
END_IF

IF SwitchDF.Q AND iFreqAdd = 120 THEN
step := 3;
END_IF


CASE step OF
	0:; (*Standby*)

	1:

		iFreqAdd := 80;
		step := 0;

	2:

		iFreqAdd := 120;
		step := 0;

	3:

		iFreqAdd := 40;
		step := 0;

END_CASE

END_FUNCTION_BLOCK

// ---- FBs/B_JKS_CustomFB/fbUltrasonicCtrl/fbUltrasonicFIFO.TcPOU
FUNCTION_BLOCK fbUltrasonicFIFO
VAR_INPUT
	bStartEnable: BOOL;

	iSourceData: INT;
	iIntervalTime_ms: INT;
END_VAR
VAR_OUTPUT
	iAverageDataCollect: INT;
END_VAR
VAR

	OnTime: TON;
	OffTime: TON;
	OnTimeRE : R_TRIG;

	Step: INT;
	StepFIFO : INT;
	FIFOFL : INT;


END_VAR

VAR_IN_OUT
	Ar10_iUltrasonic : ARRAY[1..10] OF INT;

END_VAR

(* StartEN - FIFO *)

OnTime(IN:=NOT OnTime.Q AND bStartEnable , PT:=INT_TO_TIME(iIntervalTime_ms) , Q=> , ET=> );
OnTimeRE(CLK:=OnTime.Q , Q=> );


IF OnTimeRE.Q THEN

StepFIFO:= 1;
FIFOFL := 1;
END_IF

CASE StepFIFO OF


1:
			IF FIFOFL>0 AND FIFOFL < 10 THEN

				FOR FIFOFL := 1 TO 9 DO
				Ar10_iUltrasonic[10-FIFOFL+1] := Ar10_iUltrasonic[10-FIFOFL ];
	
				END_FOR

			END_IF

IF FIFOFL >= 10 THEN
Ar10_iUltrasonic[1] := iSourceData;
StepFIFO:= 2;
END_IF

2:; (*Siap*)


99:;

END_CASE

iAverageDataCollect := (Ar10_iUltrasonic[1] + Ar10_iUltrasonic[2] + Ar10_iUltrasonic[3] + Ar10_iUltrasonic[4] + Ar10_iUltrasonic[5] + Ar10_iUltrasonic[6] + Ar10_iUltrasonic[7] + Ar10_iUltrasonic[8] + Ar10_iUltrasonic[9] + Ar10_iUltrasonic[10]) / 10 ;

END_FUNCTION_BLOCK

// ---- FBs/B_JKS_CustomFB/fbUltrasonicCtrl/fbWeberUS_AI_Conversion.TcPOU
FUNCTION_BLOCK fbWeberUS_AI_Conversion
VAR_INPUT
	iAnalogInput : INT;
	iMaxValue : INT;
	iTargetPercentage : INT;
	i1stLimitRange : INT;
	i2ndLimitRange : INT;
	tDelayTime : TIME;
	bUsActivated	 : BOOL;



END_VAR
VAR_OUTPUT
	iPercent : INT;
	b1stLimitRange : BOOL;
	b2ndLimitRange : BOOL;

END_VAR
VAR
	rPersent: REAL;
	bAnalogInEN: BOOL;
	bMaxValueEN: BOOL;
	b1stLmitRangeEN: BOOL;
	b2ndLimitRangeEN: BOOL;
	TNR: TON;
	TPR: TON;
	bTargetPEN: BOOL;
	b1stBelowRangeINT: BOOL;
	b2ndAboveRangeINT: BOOL;
	b2ndBelowRangeINT: BOOL;
	b1stAboveRangeINT: BOOL;
END_VAR
VAR // added by the converter: edge detectors and wires of the graphical bodies
    _w1 : ANY;
    _w2, _w3 : BOOL;
END_VAR

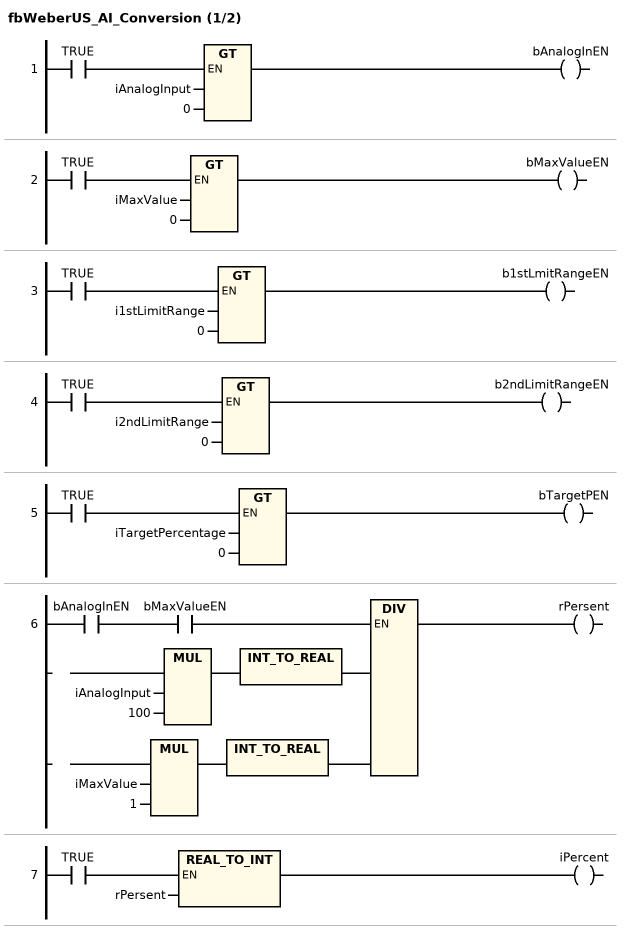
// NETWORK 1
bAnalogInEN := iAnalogInput > 0;

// NETWORK 2
bMaxValueEN := iMaxValue > 0;

// NETWORK 3
b1stLmitRangeEN := i1stLimitRange > 0;

// NETWORK 4
b2ndLimitRangeEN := i2ndLimitRange > 0;

// NETWORK 5
bTargetPEN := iTargetPercentage > 0;

// NETWORK 6
IF bAnalogInEN AND bMaxValueEN THEN _w1 := INT_TO_REAL(iAnalogInput * 100) / INT_TO_REAL(iMaxValue * 1); END_IF
rPersent := _w1;

// NETWORK 7
iPercent := REAL_TO_INT(rPersent);

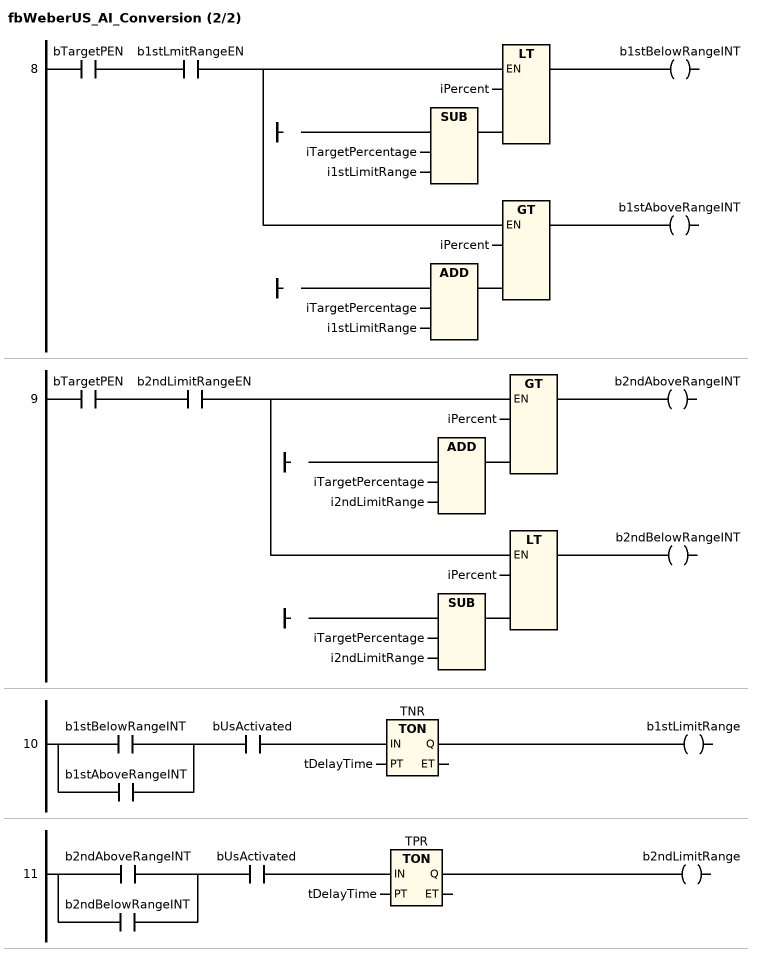
// NETWORK 8
_w2 := bTargetPEN AND b1stLmitRangeEN;
b1stBelowRangeINT := _w2 AND iPercent < iTargetPercentage - i1stLimitRange;
b1stAboveRangeINT := _w2 AND iPercent > iTargetPercentage + i1stLimitRange;

// NETWORK 9
_w3 := bTargetPEN AND b2ndLimitRangeEN;
b2ndAboveRangeINT := _w3 AND iPercent > iTargetPercentage + i2ndLimitRange;
b2ndBelowRangeINT := _w3 AND iPercent < iTargetPercentage - i2ndLimitRange;

// NETWORK 10
TNR(IN := (b1stBelowRangeINT OR b1stAboveRangeINT) AND bUsActivated, PT := tDelayTime); // TON
b1stLimitRange := TNR.Q;

// NETWORK 11
TPR(IN := (b2ndAboveRangeINT OR b2ndBelowRangeINT) AND bUsActivated, PT := tDelayTime); // TON
b2ndLimitRange := TPR.Q;

END_FUNCTION_BLOCK

// ---- FBs/B_JKS_CustomFB/fbUltrasonicCtrl/FB_WEBER.TcPOU
FUNCTION_BLOCK FB_WEBER
VAR_INPUT
	iID				: STRING;
	bStart 			: BOOL;
	bStop			: BOOL;
	bSetPoint 		: BOOL;
	iSetPoint			: INT;
	bSetFrequency 	: BOOL;
	iFrequency		: INT;
	bClk				: BOOL;
	bReset			: BOOL;
END_VAR
VAR_OUTPUT
	sCmd			: STRING;
	bBusy			: BOOL;
END_VAR
VAR
	step				: BYTE;
	R_TRIG_START			: R_TRIG;
	R_TRIG_SETFREQ 		: R_TRIG;
	R_TRIG_SETPOINT		: R_TRIG;
	R_TRIG_STOP			: R_TRIG;
END_VAR

R_TRIG_START(CLK:=bStart , Q=> );
IF R_TRIG_START.Q THEN
	step:=10;
END_IF

R_TRIG_SETPOINT(CLK:=bSetpoint , Q=> );
IF R_TRIG_SETPOINT.Q THEN
	step:=20;
END_IF

R_TRIG_STOP(CLK:=bStop , Q=> );
IF R_TRIG_STOP.Q THEN
	step:=30;
END_IF

R_TRIG_SETFREQ(CLK:=bSetFrequency , Q=> );
IF R_TRIG_SETFREQ.Q THEN
	step:=41;
END_IF


IF bClk THEN
	CASE step OF
	0:; (*Standby*)

	10:(*ON*)
		sCmd :=CONCAT( CONCAT('$$',iID),'G$R'); (*ON*)
		step:=0;

	20: (*SetPoint*)
		sCmd :=CONCAT(CONCAT(CONCAT(CONCAT('$$',iID),'R'),INT_TO_STRING(iSetPoint)),'0$R'); (*SET POINT*)
		step:=0;

	30: (*OFF*)
		sCmd :=CONCAT( CONCAT('$$',iID),'O$R'); (*ON*)
		step:=0;

	40: (*Set Frequency*)
		bBusy:=TRUE;
		sCmd :=CONCAT( CONCAT('$$',iID),'O$R'); (*OFF*)
		step:=41;

	41:
		sCmd := CONCAT(CONCAT(CONCAT(CONCAT('$$',iID),'B'),INT_TO_STRING(iFrequency)),'$R'); (*SET FREQ*)
		step:=0; (*return string base on ilD*)

	42:
		 sCmd := CONCAT(CONCAT('$$',iID),'G$R'); (*ON*)
		step:=43;

	43:
		(*bBusy:=FALSE;*)
		 sCmd := CONCAT(CONCAT(CONCAT(CONCAT('$$',iID),'R'),INT_TO_STRING(iSetPoint)),'$R'); (*SET POINT*)
		step:=0;

	51:
		sCmd := CONCAT(CONCAT(CONCAT('$$',iID),'EO'),'$R'); (*RESET ALL GENERATOR*)
		step:=0;

	END_CASE

END_IF

END_FUNCTION_BLOCK

// ---- FBs/B_JKS_CustomFB/fbUltrasonicCtrl/WeberFreqSelector.TcPOU
FUNCTION_BLOCK WeberFreqSelector
VAR_INPUT
	bSwitch : BOOL;

END_VAR
VAR_IN_OUT

	iFreqAdd : INT;


END_VAR
VAR
	SwitchDF: R_TRIG;
	step : BYTE;

END_VAR

SwitchDF (CLK:=bSwitch , Q=> );

IF iFreqAdd <> 40 AND iFreqAdd <> 80 AND iFreqAdd <> 120 THEN
iFreqAdd := 40;
END_IF

IF SwitchDF.Q AND iFreqAdd = 40 THEN
step := 1;
END_IF

IF SwitchDF.Q AND iFreqAdd = 80 THEN
step := 2;
END_IF

IF SwitchDF.Q AND iFreqAdd = 120 THEN
step := 3;
END_IF


CASE step OF
	0:; (*Standby*)

	1:

		iFreqAdd := 80;
		step := 0;

	2:

		iFreqAdd := 120;
		step := 0;

	3:

		iFreqAdd := 40;
		step := 0;

END_CASE

END_FUNCTION_BLOCK

// ---- FBs/B_JKS_CustomFB/Other/DoorOpenBasketTransfer.TcPOU
FUNCTION_BLOCK DoorOpenBasketTransfer
VAR_INPUT

	bMainOnOff:BOOL;
	bDownPost:BOOL;
	bHookPost:BOOL;
	bBasketComfirm:BOOL;

	bNextDownPost:BOOL;
	bNextUnHookPost:BOOL;



END_VAR
VAR_OUTPUT
	bBasketTransfer:BOOL;

END_VAR
VAR
	BasketTransferComplete: BOOL;
END_VAR

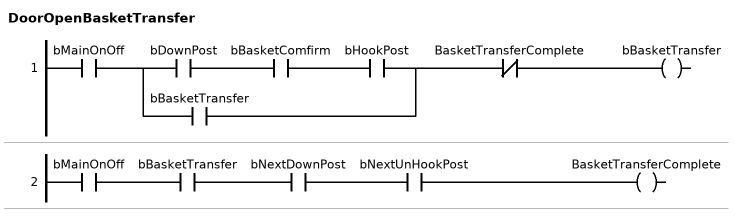
// NETWORK 1
bBasketTransfer := (bMainOnOff AND (bDownPost AND bBasketComfirm AND bHookPost OR bBasketTransfer)) AND NOT BasketTransferComplete;

// NETWORK 2
BasketTransferComplete := bMainOnOff AND bBasketTransfer AND bNextDownPost AND bNextUnHookPost;

END_FUNCTION_BLOCK

// ---- FBs/B_JKS_CustomFB/Other/fbConveyorCtrl.TcPOU
FUNCTION_BLOCK fbConveyorCtrl
VAR_INPUT
	bEnable		: BOOL;
	bRapidPB	: BOOL;
	bZone1Sensor	: BOOL;
	bZone2Sensor	: BOOL;
	bEndZoneSensor	: BOOL;
	diZone1BasketConfirmDelayTime	: DINT;
	diZone2BasketConfirmDelayTime	: DINT;
	diEndZoneBasketConfirmDelayTime	: DINT;
	diRapidPBDelayTime	: DINT;

	bLdBasketZone1MemoryBit: BOOL;
	bEmergencyStop: BOOL;
END_VAR
VAR_OUTPUT
	bMotorOnOff	: BOOL;
END_VAR
VAR
	TON1: TON;
	TRIG1: R_TRIG;
	bMotorStopBit: BOOL;
	TON2: TON;
	Trig2: R_TRIG;
	TON3: TON;
	RampIn: BOOL;
	TON4: TON;
	bConvAutoCut: BOOL;
	CVDelayOff : BOOL;
	TON5: TON;
END_VAR

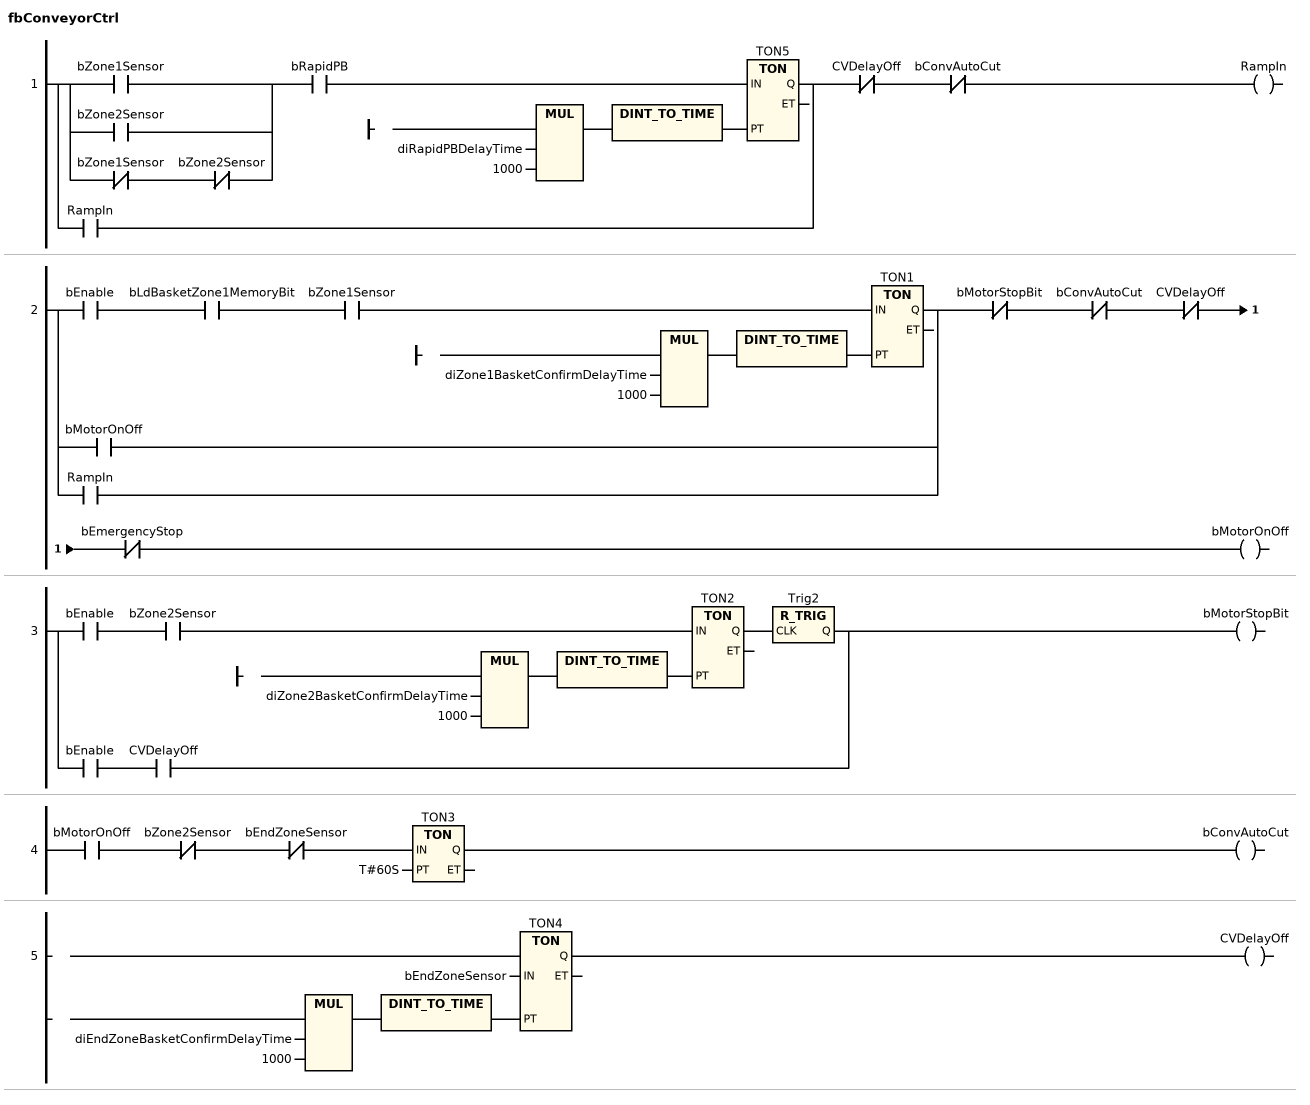
// NETWORK 1
TON5(IN := (bZone1Sensor OR bZone2Sensor OR NOT bZone1Sensor AND NOT bZone2Sensor) AND bRapidPB, PT := DINT_TO_TIME(diRapidPBDelayTime * 1000)); // TON
RampIn := (TON5.Q OR RampIn) AND NOT CVDelayOff AND NOT bConvAutoCut;

// NETWORK 2
TON1(IN := bEnable AND bLdBasketZone1MemoryBit AND bZone1Sensor, PT := DINT_TO_TIME(diZone1BasketConfirmDelayTime * 1000)); // TON
bMotorOnOff := (TON1.Q OR bMotorOnOff OR RampIn) AND NOT bMotorStopBit AND NOT bConvAutoCut AND NOT CVDelayOff AND NOT bEmergencyStop;

// NETWORK 3
TON2(IN := bEnable AND bZone2Sensor, PT := DINT_TO_TIME(diZone2BasketConfirmDelayTime * 1000)); // TON
Trig2(CLK := TON2.Q); // R_TRIG
bMotorStopBit := Trig2.Q OR bEnable AND CVDelayOff;

// NETWORK 4
TON3(IN := bMotorOnOff AND NOT bZone2Sensor AND NOT bEndZoneSensor, PT := T#60S); // TON
bConvAutoCut := TON3.Q;

// NETWORK 5
TON4(IN := bEndZoneSensor, PT := DINT_TO_TIME(diEndZoneBasketConfirmDelayTime * 1000)); // TON
CVDelayOff := TON4.Q;

END_FUNCTION_BLOCK

// ---- FBs/B_JKS_CustomFB/Other/fbIndirectAddStringArray.TcPOU
FUNCTION_BLOCK fbIndirectAddStringArray
VAR_INPUT
	bSavePB : BOOL;
	bLoadPB : BOOL;
	iProgramNo : INT;

END_VAR
VAR_OUTPUT PERSISTENT

	bSaveInd : BOOL;
	bLoadInd : BOOL;
	AR99sStringData1 : ARRAY[0..99] OF STRING;
	AR99sStringData2 : ARRAY[0..99] OF STRING;

END_VAR


VAR_IN_OUT

	sString1 : STRING;
	sString2 : STRING;

END_VAR

VAR
	SaveTimerDelay: TON;
	SaveIndHR: BOOL;
	LoadIndHR: BOOL;
	LoadTimerDelay: TON;
	SelfCheck: BOOL;
	SelfCheckTimer: TON;
	PreviousProgram: INT;
	SelfCheckLoop: BOOL;
	bLoadEN: BOOL;
	LoadDF: R_TRIG;
	LoadENDF: R_TRIG;
	SaveDF: R_TRIG;
END_VAR

(*Save Indicator*)
IF bSavePB THEN
SaveIndHR := TRUE;
END_IF

SaveTimerDelay(IN:=SaveIndHR, PT:=T#1s, Q=>, ET=> );
IF SaveTimerDelay.Q THEN
SaveIndHR := FALSE;
END_IF

IF SaveIndHR AND NOT SaveTimerDelay.Q THEN
bSaveInd := TRUE;
ELSE
bSaveInd := FALSE;
END_IF

(*Load Indicator*)
IF bLoadPB THEN
LoadIndHR := TRUE;
END_IF

LoadTimerDelay(IN:=LoadIndHR, PT:=T#1s, Q=>, ET=> );
IF LoadTimerDelay.Q THEN
LoadIndHR := FALSE;
END_IF

IF LoadIndHR AND NOT LoadTimerDelay.Q THEN
bLoadInd := TRUE;
ELSE
bLoadInd := FALSE;
END_IF

(*Self Check of Program No Change*)

SelfCheckTimer(IN:=NOT SelfCheckLoop, PT:=T#0.5s, Q=>, ET=> );

	IF SelfCheckTimer.Q THEN
	PreviousProgram := iProgramNo ;
	SelfCheckLoop := TRUE;
	ELSE
	SelfCheckLoop := FALSE;
	END_IF

IF iProgramNo <> PreviousProgram THEN
bLoadEN := TRUE;
ELSE
bLoadEN := FALSE;
END_IF

(*Recipe Load*)
LoadDF(CLK:=bLoadPB, Q=> );
LoadENDF (CLK:=bLoadEN, Q=> );

IF LoadDF.Q OR LoadENDF.Q THEN
sString1 := AR99sStringData1[iProgramNo];
sString2 := AR99sStringData2[iProgramNo];
END_IF

(*Recipe Save*)
SaveDF(CLK:=bSavePB, Q=> );

IF SaveDF.Q THEN
AR99sStringData1[iProgramNo] := sString1;
AR99sStringData2[iProgramNo] := sString2;
END_IF

END_FUNCTION_BLOCK

// ---- FBs/B_JKS_CustomFB/Other/fbKeyConversionBarKpa.TcPOU
FUNCTION_BLOCK fbKeyConversionBarKpa
VAR_INPUT
	bEN : BOOL;
	iRaw : INT;
(*	rKpaRatio : REAL;
	rBarRatio : REAL;
*)	bZeroReset : BOOL;
	tRefreshTime: TIME;


END_VAR
VAR_OUTPUT
	rKpaResult : REAL;
	rBarResult : REAL;
END_VAR


VAR PERSISTENT



END_VAR
VAR PERSISTENT
	iDelta: INT;
	iRawAverage: ARRAY [1..20] OF INT;
	FIFODone : R_TRIG;
	iAveAdd: INT;
	iTotal: DINT;
	iAveRaw: INT;
	iAveRawINT: DINT;
	rKpaResultINT: REAL;
	rBarResultINT: REAL;
END_VAR
VAR
	FIFOFL: INT;
	ClockPulse: TON;

END_VAR

ClockPulse(IN:=NOT ClockPulse.Q , PT:=tRefreshTime , Q=> , ET=> );

IF ClockPulse.Q THEN
FIFOFL := 1;
END_IF

IF FIFOFL < 20+1 THEN

	FOR FIFOFL := 1 TO 20 DO
	iRawAverage[FIFOFL] := iRawAverage[FIFOFL+1];
	END_FOR

END_IF

(*FIFODone(CLK:= FIFOFL > 20 , Q=> );*)

IF  ClockPulse.Q THEN
iRawAverage[20] := iRaw;
iTotal := 0;
iAveAdd := 1;

	FOR iAveAdd := 1 TO 20 DO
	iTotal := iTotal + iRawAverage[iAveAdd];
	END_FOR

iAveRawINT := iTotal / 20 ;
iAveRaw := DINT_TO_INT(iAveRawINT);


END_IF


IF bEN THEN

	IF bEN THEN
	rKpaResultINT := (INT_TO_REAL(iRaw)/(13106.8/5))-101.3;
(*	ELSE
	rKpaResult := (INT_TO_REAL(iAveRaw-iDelta)/(32767/1114.3))-101.3;*)
	END_IF

	IF bEN THEN
	rBarResultINT := (INT_TO_REAL(iAveRaw-iDelta)/(32767/11))-1;
(*	ELSE
	rKpaResult := 0;*)
	END_IF

	IF rKpaResultINT >= -101.3 THEN
	rKpaResult := rKpaResultINT;
	ELSE
	rKpaResult := -101.3;
	END_IF

	IF rKpaResultINT >= -1 THEN
	rBarResult := rBarResultINT;
	ELSE
	rBarResult := -1;
	END_IF


ELSE

rKpaResult := 0;
rBarResult := 0;
END_IF

IF bZeroReset THEN
;	(*iDelta := (iAveRaw-(32767/11));*)
END_IF

END_FUNCTION_BLOCK

// ---- FBs/B_JKS_CustomFB/Other/fbLdConveyor3Zones.TcPOU
FUNCTION_BLOCK fbLdConveyor3Zones
VAR_INPUT

	bEnable		: BOOL;
	bRapidPB	: BOOL;
	bLdBasketZone1TransferMemoryBit: BOOL;
	bLdBasketZone1ConfirmMemoryBit: BOOL;
	bLdBasketZone2TransferMemoryBit: BOOL;
	bLdBasketZone2ConfirmMemoryBit	: BOOL;

	bLdSensor1: BOOL;
	bLdSensor2: BOOL;
	bLdEndSensor: BOOL;

	diZone1BasketConfirmDelayTime	: DINT;

(*	diZone2BasketConfirmDelayTime	: DINT;
	diRapidPBDelayTime	: DINT;
*)
	diEndZoneBasketConfirmDelayTime	: DINT;

	bEmergencyStop: BOOL;
END_VAR
VAR_OUTPUT
	bMotorOnOff	: BOOL;
END_VAR
VAR
	bRapidPBRE: R_TRIG;
	bMotorStopBit: BOOL;
	TON1: TON;
	TON2: TON;
	bConvAutoCut: BOOL;
	tLdZone1SensorDelayTime: TON;

	(*TRIG1: R_TRIG;
	Trig2: R_TRIG;
	TON3: TON;
	RampIn: BOOL;
	TON4: TON;
	CVDelayOff : BOOL;
	TON5: TON;*)

END_VAR

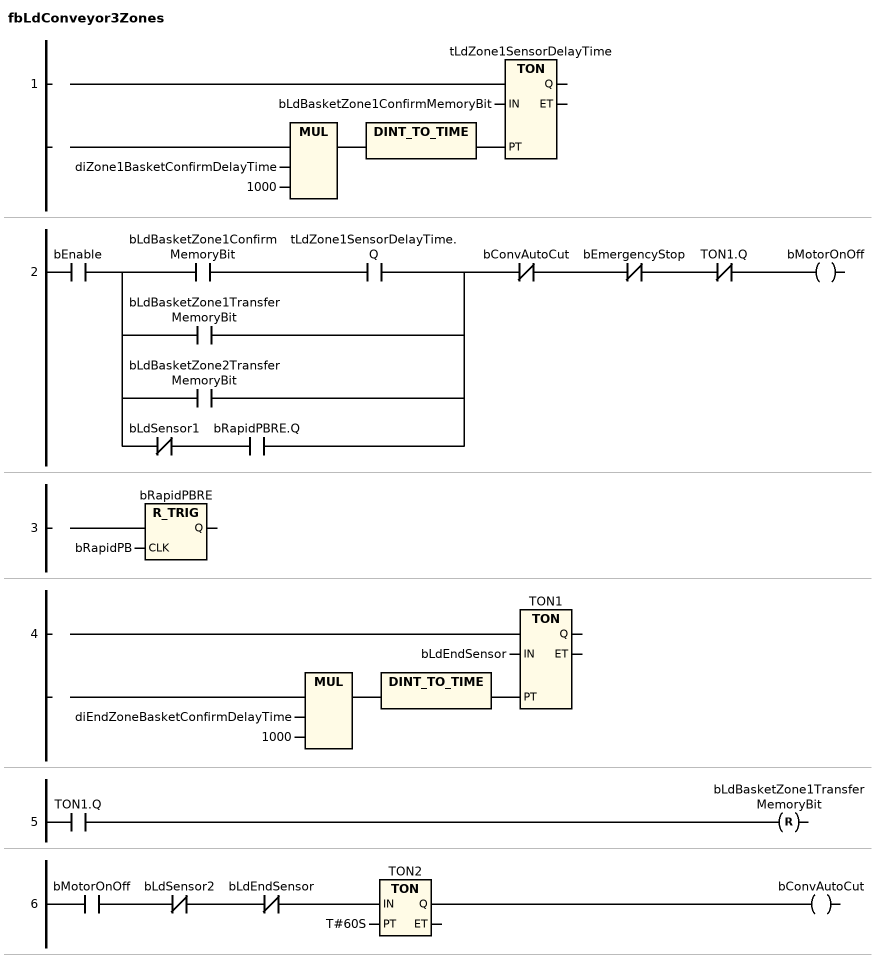
// NETWORK 1
tLdZone1SensorDelayTime(IN := bLdBasketZone1ConfirmMemoryBit, PT := DINT_TO_TIME(diZone1BasketConfirmDelayTime * 1000)); // TON

// NETWORK 2
bMotorOnOff := (bEnable AND (bLdBasketZone1ConfirmMemoryBit AND tLdZone1SensorDelayTime.Q OR bLdBasketZone1TransferMemoryBit OR bLdBasketZone2TransferMemoryBit OR NOT bLdSensor1 AND bRapidPBRE.Q)) AND NOT bConvAutoCut AND NOT bEmergencyStop AND NOT TON1.Q;

// NETWORK 3
bRapidPBRE(CLK := bRapidPB); // R_TRIG

// NETWORK 4
TON1(IN := bLdEndSensor, PT := DINT_TO_TIME(diEndZoneBasketConfirmDelayTime * 1000)); // TON

// NETWORK 5
bLdBasketZone1TransferMemoryBit R= TON1.Q;

// NETWORK 6
TON2(IN := bMotorOnOff AND NOT bLdSensor2 AND NOT bLdEndSensor, PT := T#60S); // TON
bConvAutoCut := TON2.Q;

END_FUNCTION_BLOCK

// ---- FBs/B_JKS_CustomFB/Other/fbLoadingConveyor3Zones.TcPOU
PROGRAM fbLoadingConveyor3Zones
VAR
	bEnable: BOOL;
	bLd1ConfirmAvailable: BOOL;
	bLd1TransferAvailable: BOOL;

	bLd2ConfirmAvailable: BOOL;
	bLd2TransferAvailable: BOOL;

	bLd3ConfirmAvailable: BOOL;
	bLd3TransferAvailable: BOOL;

	bLdSensor1: BOOL;
	bLdSensor2: BOOL;
	bLdSensor3: BOOL;

	bRapidPB : BOOL;

	bBarcodeValid: BOOL;

	bMotor: BOOL;


	tLdSensor1OffDelay: TON;
	bMotorRE: R_TRIG;
	bMotorFE: F_TRIG;
	bLdSensor1RE: R_TRIG;
	bLdSensor2RE: R_TRIG;
	bLdSensor3RE: R_TRIG;
	bBarcodeValidRE: R_TRIG;
	bRapidPBRE: R_TRIG;
	tLdSensor3OnDelay: TON;
	tLdSensor3withMotorOnDelay: TON;
END_VAR

(*Rising Edge*)
bMotorRE(CLK:=bMotor , Q=> );
bLdSensor1RE(CLK:=bLdSensor1 , Q=> );
bLdSensor2RE(CLK:=bLdSensor2 , Q=> );
bLdSensor3RE(CLK:=bLdSensor3 , Q=> );
bBarcodeValidRE(CLK:=bBarcodeValid , Q=> );
bRapidPBRE(CLK:=bRapidPB , Q=> );

(*Falling Edge*)
bMotorFE(CLK:=bMotor , Q=> );



(*Loading Sequence*)

tLdSensor3OnDelay(IN:=bLdSensor3  , PT:=t#3s , Q=> , ET=> );

IF tLdSensor3OnDelay.Q THEN
	bLd1TransferAvailable := FALSE;
END_IF


IF bEnable THEN

	IF (bLd1ConfirmAvailable OR bLd1TransferAvailable OR bLd2TransferAvailable OR (NOT bLdSensor1 AND bRapidPBRE.Q))  AND NOT tLdSensor3OnDelay.Q THEN
	bMotor := TRUE;
	ELSE
	bMotor := FALSE;
	END_IF


ELSE

	bMotor := FALSE;

END_IF


(*Basket Memory Control*)

tLdSensor1OffDelay(IN:=NOT bLdSensor1 , PT:=t#2s , Q=> , ET=> );

IF bLdSensor1 AND bBarcodeValidRE.Q THEN
bLd1ConfirmAvailable := TRUE;
END_IF

IF tLdSensor1OffDelay.Q THEN
bLd1ConfirmAvailable := FALSE;
END_IF

(*Confirm to Transfer*)
IF bMotorRE.Q AND bLd1ConfirmAvailable THEN
bLd1TransferAvailable := TRUE;
bLd1ConfirmAvailable := FALSE;
END_IF

IF bMotorRE.Q AND bLd2ConfirmAvailable THEN
bLd2TransferAvailable := TRUE;
bLd2ConfirmAvailable := FALSE;
END_IF

(*Transfer to Confirm*)
IF bLdSensor2RE.Q AND bLd1TransferAvailable THEN
bLd2ConfirmAvailable := TRUE;
bLd1TransferAvailable := FALSE;
END_IF

IF bLdSensor3RE.Q AND bLd2TransferAvailable THEN
bLd3ConfirmAvailable := TRUE;
bLd2TransferAvailable := FALSE;
END_IF

END_PROGRAM

// ---- FBs/B_JKS_CustomFB/Other/fbMultipleArmBasketMemory.TcPOU
FUNCTION_BLOCK fbMultipleArmBasketMemory
VAR_INPUT
END_VAR
VAR_OUTPUT
END_VAR
VAR
END_VAR

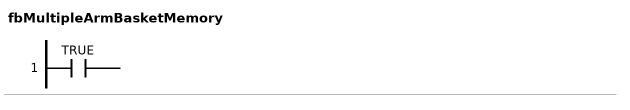
// NETWORK 1

END_FUNCTION_BLOCK

// ---- FBs/B_JKS_CustomFB/Other/fbPX3524ConversionBarKpa.TcPOU
FUNCTION_BLOCK fbPX3524ConversionBarKpa
VAR_INPUT
	bEN : BOOL;
	iRaw : INT;
(*	rKpaRatio : REAL;
	rBarRatio : REAL;
*)	bZeroReset : BOOL;
	tRefreshTime: TIME;


END_VAR
VAR_OUTPUT
	rKpaResult : REAL;
	rBarResult : REAL;
END_VAR


VAR PERSISTENT



END_VAR
VAR PERSISTENT
	iDelta: INT;
	iRawAverage: ARRAY [1..20] OF INT;
	FIFODone : R_TRIG;
	iAveAdd: INT;
	iTotal: DINT;
	iAveRaw: INT;
	iAveRawINT: DINT;
	rKpaResultINT: REAL;
	rBarResultINT: REAL;
END_VAR
VAR
	FIFOFL: INT;
	ClockPulse: TON;

END_VAR

ClockPulse(IN:=NOT ClockPulse.Q , PT:=tRefreshTime , Q=> , ET=> );

IF ClockPulse.Q THEN
FIFOFL := 1;
END_IF

IF FIFOFL < 20+1 THEN

	FOR FIFOFL := 1 TO 20 DO
	iRawAverage[FIFOFL] := iRawAverage[FIFOFL+1];
	END_FOR

END_IF

(*FIFODone(CLK:= FIFOFL > 20 , Q=> );*)

IF  ClockPulse.Q THEN
iRawAverage[20] := iRaw;
iTotal := 0;
iAveAdd := 1;

	FOR iAveAdd := 1 TO 20 DO
	iTotal := iTotal + iRawAverage[iAveAdd];
	END_FOR

iAveRawINT := iTotal / 20 ;
iAveRaw := DINT_TO_INT(iAveRawINT);


END_IF


IF bEN THEN

	IF bEN THEN
	rKpaResultINT := (INT_TO_REAL(iRaw)/(32767/1114.3))-101.3;
(*	ELSE
	rKpaResult := (INT_TO_REAL(iAveRaw-iDelta)/(32767/1114.3))-101.3;*)
	END_IF

	IF bEN THEN
	rBarResultINT := (INT_TO_REAL(iAveRaw-iDelta)/(32767/11))-1;
(*	ELSE
	rKpaResult := 0;*)
	END_IF

	IF rKpaResultINT >= -101.3 THEN
	rKpaResult := rKpaResultINT;
	ELSE
	rKpaResult := -101.3;
	END_IF

	IF rKpaResultINT >= -1 THEN
	rBarResult := rBarResultINT;
	ELSE
	rBarResult := -1;
	END_IF


ELSE

rKpaResult := 0;
rBarResult := 0;
END_IF

IF bZeroReset THEN
;	(*iDelta := (iAveRaw-(32767/11));*)
END_IF

END_FUNCTION_BLOCK

// ---- FBs/B_JKS_CustomFB/Other/fbStnRecipeWithSubAndCall.TcPOU
FUNCTION_BLOCK fbStnRecipeWithSubAndCall
VAR_INPUT
	bSavePB : BOOL;
	bLoadPB : BOOL;



END_VAR

VAR_OUTPUT PERSISTENT

	bSaveInd : BOOL;
	bLoadInd : BOOL;

	iSeqCallPresentProgram1 : INT;
	iSeqCallPresentProgram2 : INT;
	iSeqCallPresentProgram3 : INT;
	iSeqCallPresentProgram4 : INT;
	iSeqCallPresentProgram5 : INT;
	iSeqCallPresentProgram6 : INT;
	iSeqCallPresentProgram7 : INT;
	iSeqCallPresentProgram8 : INT;
	iSeqCallPresentProgram9 : INT;
	iSeqCallPresentProgram10 : INT;

	iCallSubProAdd1 : INT;
	iCallSubProAdd2 : INT;
	iCallSubProAdd3 : INT;
	iCallSubProAdd4 : INT;
	iCallSubProAdd5 : INT;
	iCallSubProAdd6 : INT;
	iCallSubProAdd7 : INT;
	iCallSubProAdd8 : INT;
	iCallSubProAdd9 : INT;
	iCallSubProAdd10 : INT;
	iCallRecipeTotalTime : INT;
	AR10_iCallSubProTotalTime : ARRAY[1..10] OF INT;

END_VAR

VAR_IN_OUT PERSISTENT

	iMainNo : INT;
	iSequencePresentProgram1 : INT;
	iSequencePresentProgram2 : INT;
	iSequencePresentProgram3 : INT;
	iSequencePresentProgram4 : INT;
	iSequencePresentProgram5 : INT;
	iSequencePresentProgram6 : INT;
	iSequencePresentProgram7 : INT;
	iSequencePresentProgram8 : INT;
	iSequencePresentProgram9 : INT;
	iSequencePresentProgram10 : INT;



	iSubNo : INT;
	iSubProAdd1 : INT;
	iSubProAdd2 : INT;
	iSubProAdd3 : INT;
	iSubProAdd4 : INT;
	iSubProAdd5 : INT;
	iSubProAdd6 : INT;
	iSubProAdd7 : INT;
	iSubProAdd8 : INT;
	iSubProAdd9 : INT;
	iSubProAdd10 : INT;
	iCallMainRecipeNo : INT;
	iCallSubRecipeNo : INT;
	iTotalTimeMainRecipeNo : INT;
	iTotalTimeSubRecipeNo : INT;




END_VAR

VAR PERSISTENT

	AR200iInterger1 : ARRAY[0..200] OF INT;
	AR200iInterger2 : ARRAY[0..200] OF INT;
	AR200iInterger3 : ARRAY[0..200] OF INT;
	AR200iInterger4 : ARRAY[0..200] OF INT;
	AR200iInterger5 : ARRAY[0..200] OF INT;
	AR200iInterger6 : ARRAY[0..200] OF INT;
	AR200iInterger7 : ARRAY[0..200] OF INT;
	AR200iInterger8 : ARRAY[0..200] OF INT;
	AR200iInterger9 : ARRAY[0..200] OF INT;
	AR200iInterger10 : ARRAY[0..200] OF INT;
	AR200iInterger11 : ARRAY[0..200] OF INT;
	AR200iInterger12 : ARRAY[0..200] OF INT;
	AR200iInterger13 : ARRAY[0..200] OF INT;
	AR200iInterger14 : ARRAY[0..200] OF INT;
	AR200iInterger15 : ARRAY[0..200] OF INT;
	AR200iInterger16 : ARRAY[0..200] OF INT;
	AR200iInterger17 : ARRAY[0..200] OF INT;
	AR200iInterger18 : ARRAY[0..200] OF INT;
	AR200iInterger19 : ARRAY[0..200] OF INT;
	AR200iInterger20 : ARRAY[0..200] OF INT;
	AR200iInterger21 : ARRAY[0..200] OF INT;
	AR200iInterger22 : ARRAY[0..200] OF INT;
	AR200iInterger23 : ARRAY[0..200] OF INT;
	AR200iInterger24 : ARRAY[0..200] OF INT;
	AR200iInterger25 : ARRAY[0..200] OF INT;
	AR200iInterger26 : ARRAY[0..200] OF INT;
	AR200iInterger27 : ARRAY[0..200] OF INT;
	AR200iInterger28 : ARRAY[0..200] OF INT;
	AR200iInterger29 : ARRAY[0..200] OF INT;
	AR200iInterger30 : ARRAY[0..200] OF INT;
	AR200iInterger31 : ARRAY[0..200] OF INT;
	AR200iInterger32 : ARRAY[0..200] OF INT;
	AR200iInterger33 : ARRAY[0..200] OF INT;
	AR200iInterger34 : ARRAY[0..200] OF INT;
	AR200iInterger35 : ARRAY[0..200] OF INT;
	AR200iInterger36 : ARRAY[0..200] OF INT;
	AR200iInterger37 : ARRAY[0..200] OF INT;
	AR200iInterger38 : ARRAY[0..200] OF INT;
	AR200iInterger39 : ARRAY[0..200] OF INT;
	AR200iInterger40 : ARRAY[0..200] OF INT;
	AR200iInterger41 : ARRAY[0..200] OF INT;
	AR200iInterger42 : ARRAY[0..200] OF INT;
	AR200iInterger43 : ARRAY[0..200] OF INT;
	AR200iInterger44 : ARRAY[0..200] OF INT;
	AR200iInterger45 : ARRAY[0..200] OF INT;
	AR200iInterger46 : ARRAY[0..200] OF INT;
	AR200iInterger47 : ARRAY[0..200] OF INT;
	AR200iInterger48 : ARRAY[0..200] OF INT;
	AR200iInterger49 : ARRAY[0..200] OF INT;
	AR200iInterger50 : ARRAY[0..200] OF INT;
	AR200iInterger51 : ARRAY[0..200] OF INT;
	AR200iInterger52 : ARRAY[0..200] OF INT;
	AR200iInterger53 : ARRAY[0..200] OF INT;
	AR200iInterger54 : ARRAY[0..200] OF INT;
	AR200iInterger55 : ARRAY[0..200] OF INT;
	AR200iInterger56 : ARRAY[0..200] OF INT;
	AR200iInterger57 : ARRAY[0..200] OF INT;
	AR200iInterger58 : ARRAY[0..200] OF INT;
	AR200iInterger59 : ARRAY[0..200] OF INT;
	AR200iInterger60 : ARRAY[0..200] OF INT;
	AR200iInterger61 : ARRAY[0..200] OF INT;
	AR200iInterger62 : ARRAY[0..200] OF INT;
	AR200iInterger63 : ARRAY[0..200] OF INT;
	AR200iInterger64 : ARRAY[0..200] OF INT;
	AR200iInterger65 : ARRAY[0..200] OF INT;
	AR200iInterger66 : ARRAY[0..200] OF INT;
	AR200iInterger67 : ARRAY[0..200] OF INT;
	AR200iInterger68 : ARRAY[0..200] OF INT;
	AR200iInterger69 : ARRAY[0..200] OF INT;
	AR200iInterger70 : ARRAY[0..200] OF INT;
	AR200iInterger71 : ARRAY[0..200] OF INT;
	AR200iInterger72 : ARRAY[0..200] OF INT;
	AR200iInterger73 : ARRAY[0..200] OF INT;
	AR200iInterger74 : ARRAY[0..200] OF INT;
	AR200iInterger75 : ARRAY[0..200] OF INT;
	AR200iInterger76 : ARRAY[0..200] OF INT;
	AR200iInterger77 : ARRAY[0..200] OF INT;
	AR200iInterger78 : ARRAY[0..200] OF INT;
	AR200iInterger79 : ARRAY[0..200] OF INT;
	AR200iInterger80 : ARRAY[0..200] OF INT;
	AR200iInterger81 : ARRAY[0..200] OF INT;
	AR200iInterger82 : ARRAY[0..200] OF INT;
	AR200iInterger83 : ARRAY[0..200] OF INT;
	AR200iInterger84 : ARRAY[0..200] OF INT;
	AR200iInterger85 : ARRAY[0..200] OF INT;
	AR200iInterger86 : ARRAY[0..200] OF INT;
	AR200iInterger87 : ARRAY[0..200] OF INT;
	AR200iInterger88 : ARRAY[0..200] OF INT;
	AR200iInterger89 : ARRAY[0..200] OF INT;
	AR200iInterger90 : ARRAY[0..200] OF INT;
	AR200iInterger91 : ARRAY[0..200] OF INT;
	AR200iInterger92 : ARRAY[0..200] OF INT;
	AR200iInterger93 : ARRAY[0..200] OF INT;
	AR200iInterger94 : ARRAY[0..200] OF INT;
	AR200iInterger95 : ARRAY[0..200] OF INT;
	AR200iInterger96 : ARRAY[0..200] OF INT;
	AR200iInterger97 : ARRAY[0..200] OF INT;
	AR200iInterger98 : ARRAY[0..200] OF INT;
	AR200iInterger99 : ARRAY[0..200] OF INT;
	AR200iInterger100 : ARRAY[0..200] OF INT;

	AR200iInterger101 : ARRAY[0..200] OF INT;
	AR200iInterger102 : ARRAY[0..200] OF INT;
	AR200iInterger103 : ARRAY[0..200] OF INT;
	AR200iInterger104 : ARRAY[0..200] OF INT;
	AR200iInterger105 : ARRAY[0..200] OF INT;
	AR200iInterger106 : ARRAY[0..200] OF INT;
	AR200iInterger107 : ARRAY[0..200] OF INT;
	AR200iInterger108 : ARRAY[0..200] OF INT;
	AR200iInterger109 : ARRAY[0..200] OF INT;
	AR200iInterger110 : ARRAY[0..200] OF INT;

	AR200iTotalTimeIntCall : ARRAY[1..200] OF INT;

	iSeqCallTTPresentProgram1 : INT;
	iSeqCallTTPresentProgram2 : INT;
	iSeqCallTTPresentProgram3 : INT;
	iSeqCallTTPresentProgram4 : INT;
	iSeqCallTTPresentProgram5 : INT;
	iSeqCallTTPresentProgram6 : INT;
	iSeqCallTTPresentProgram7 : INT;
	iSeqCallTTPresentProgram8 : INT;
	iSeqCallTTPresentProgram9 : INT;
	iSeqCallTTPresentProgram10 : INT;

	AR200iIntCall : ARRAY[1..200] OF INT;
	AR200iInt : ARRAY[1..200] OF INT;

END_VAR

VAR

	SaveIndHr: BOOL;
	SaveTimerDelay: TON;
	LoadIndHr: BOOL;
	LoadTimerDelay: TON;
	SelfCheckTimer: TON;
	SelfCheckloop: BOOL;
	LoadDF: R_TRIG;
	LoadENDF: R_TRIG;
	SaveDF: R_TRIG;

	i: INT;
	Partvalid: BOOL;

	SubLoadENDF: R_TRIG;
	SelfCheckSubTimer: TON;
	SelfCheckSubloop: BOOL;


	PreviousNo: INT;
	PreviousSubNo: INT;
	bLoadEn: BOOL;
	bSubLoadEN: BOOL;


	iTotalTimeMainRecipeNoRE : R_TRIG;
	ScanTTFL : INT;

	bStartTTScan: BOOL;
END_VAR

IF iMainNo < 1 THEN
iMainNo := 1;
END_IF

IF iMainNo > 99 THEN
iMainNo := 99;
END_IF

IF iSubNo < 1 THEN
iSubNo := 1;
END_IF

IF iSubNo > 10 THEN
iSubNo := 10;
END_IF
(*
IF iCallMainRecipeNo < 1 THEN
iCallMainRecipeNo := 1;
END_IF

IF iCallMainRecipeNo > 99 THEN
iCallMainRecipeNo := 99;
END_IF

IF iCallSubRecipeNo < 1 THEN
iCallSubRecipeNo := 1;
END_IF

IF iCallSubRecipeNo > 10 THEN
iCallSubRecipeNo := 10;
END_IF
*)

IF bSavePB THEN
SaveIndHr := TRUE;
END_IF

SaveTimerDelay(IN:=SaveIndHr, PT := T#1s, Q=>, ET=>);
IF SaveTimerDelay.Q THEN
SaveIndHr := FALSE;
END_IF

IF SaveIndHr AND NOT SaveTimerDelay.Q THEN
bSaveInd := TRUE;
ELSE
bSaveInd := FALSE;
END_IF

IF bLoadPB THEN
LoadIndHr := TRUE;
END_IF

LoadTimerDelay(IN:=LoadIndHr, PT := T#1s, Q=>, ET=>);
IF loadtimerdelay.Q THEN
LoadIndHr := FALSE;
END_IF

IF loadIndHr AND NOT LoadTimerDelay.Q THEN
bLoadInd := TRUE;
ELSE
bLoadInd := FALSE;
END_IF

SelfCheckTimer(IN:=NOT SelfCheckloop, PT := T#0.5s, Q=>, ET=>);

	IF SelfCheckTimer.Q THEN
	PreviousNo := iMainNo;
	SelfCheckloop := TRUE;
	ELSE
	SelfCheckloop := FALSE;
	END_IF

IF iMainNo <> PreviousNo THEN
bLoadEn := TRUE;
ELSE
bLoadEn := FALSE;
END_IF


SelfCheckSubTimer(IN:=NOT SelfCheckSubloop, PT := T#0.5s, Q=>, ET=>);

	IF SelfCheckTimer.Q THEN
	PreviousSubNo := iSubNo;
	SelfCheckSubloop := TRUE;
	ELSE
	SelfCheckSubloop := FALSE;
	END_IF

IF iSubNo <> PreviousSubNo THEN
bSubLoadEN := TRUE;
ELSE
bSubLoadEN := FALSE;
END_IF



LoadDF(CLK:=bLoadPB OR bLoadEn OR bSubLoadEN ,Q=>);

IF LoadDF.Q THEN


AR200iInt[1] := AR200iInterger1[iMainNo];
AR200iInt[2] := AR200iInterger2[iMainNo];
AR200iInt[3] := AR200iInterger3[iMainNo];
AR200iInt[4] := AR200iInterger4[iMainNo];
AR200iInt[5] := AR200iInterger5[iMainNo];
AR200iInt[6] := AR200iInterger6[iMainNo];
AR200iInt[7] := AR200iInterger7[iMainNo];
AR200iInt[8] := AR200iInterger8[iMainNo];
AR200iInt[9] := AR200iInterger9[iMainNo];
AR200iInt[10] := AR200iInterger10[iMainNo];
AR200iInt[11] := AR200iInterger11[iMainNo];
AR200iInt[12] := AR200iInterger12[iMainNo];
AR200iInt[13] := AR200iInterger13[iMainNo];
AR200iInt[14] := AR200iInterger14[iMainNo];
AR200iInt[15] := AR200iInterger15[iMainNo];
AR200iInt[16] := AR200iInterger16[iMainNo];
AR200iInt[17] := AR200iInterger17[iMainNo];
AR200iInt[18] := AR200iInterger18[iMainNo];
AR200iInt[19] := AR200iInterger19[iMainNo];
AR200iInt[20] := AR200iInterger20[iMainNo];
AR200iInt[21] := AR200iInterger21[iMainNo];
AR200iInt[22] := AR200iInterger22[iMainNo];
AR200iInt[23] := AR200iInterger23[iMainNo];
AR200iInt[24] := AR200iInterger24[iMainNo];
AR200iInt[25] := AR200iInterger25[iMainNo];
AR200iInt[26] := AR200iInterger26[iMainNo];
AR200iInt[27] := AR200iInterger27[iMainNo];
AR200iInt[28] := AR200iInterger28[iMainNo];
AR200iInt[29] := AR200iInterger29[iMainNo];
AR200iInt[30] := AR200iInterger30[iMainNo];
AR200iInt[31] := AR200iInterger31[iMainNo];
AR200iInt[32] := AR200iInterger32[iMainNo];
AR200iInt[33] := AR200iInterger33[iMainNo];
AR200iInt[34] := AR200iInterger34[iMainNo];
AR200iInt[35] := AR200iInterger35[iMainNo];
AR200iInt[36] := AR200iInterger36[iMainNo];
AR200iInt[37] := AR200iInterger37[iMainNo];
AR200iInt[38] := AR200iInterger38[iMainNo];
AR200iInt[39] := AR200iInterger39[iMainNo];
AR200iInt[40] := AR200iInterger40[iMainNo];
AR200iInt[41] := AR200iInterger41[iMainNo];
AR200iInt[42] := AR200iInterger42[iMainNo];
AR200iInt[43] := AR200iInterger43[iMainNo];
AR200iInt[44] := AR200iInterger44[iMainNo];
AR200iInt[45] := AR200iInterger45[iMainNo];
AR200iInt[46] := AR200iInterger46[iMainNo];
AR200iInt[47] := AR200iInterger47[iMainNo];
AR200iInt[48] := AR200iInterger48[iMainNo];
AR200iInt[49] := AR200iInterger49[iMainNo];
AR200iInt[50] := AR200iInterger50[iMainNo];
AR200iInt[51] := AR200iInterger51[iMainNo];
AR200iInt[52] := AR200iInterger52[iMainNo];
AR200iInt[53] := AR200iInterger53[iMainNo];
AR200iInt[54] := AR200iInterger54[iMainNo];
AR200iInt[55] := AR200iInterger55[iMainNo];
AR200iInt[56] := AR200iInterger56[iMainNo];
AR200iInt[57] := AR200iInterger57[iMainNo];
AR200iInt[58] := AR200iInterger58[iMainNo];
AR200iInt[59] := AR200iInterger59[iMainNo];
AR200iInt[60] := AR200iInterger60[iMainNo];
AR200iInt[61] := AR200iInterger61[iMainNo];
AR200iInt[62] := AR200iInterger62[iMainNo];
AR200iInt[63] := AR200iInterger63[iMainNo];
AR200iInt[64] := AR200iInterger64[iMainNo];
AR200iInt[65] := AR200iInterger65[iMainNo];
AR200iInt[66] := AR200iInterger66[iMainNo];
AR200iInt[67] := AR200iInterger67[iMainNo];
AR200iInt[68] := AR200iInterger68[iMainNo];
AR200iInt[69] := AR200iInterger69[iMainNo];
AR200iInt[70] := AR200iInterger70[iMainNo];
AR200iInt[71] := AR200iInterger71[iMainNo];
AR200iInt[72] := AR200iInterger72[iMainNo];
AR200iInt[73] := AR200iInterger73[iMainNo];
AR200iInt[74] := AR200iInterger74[iMainNo];
AR200iInt[75] := AR200iInterger75[iMainNo];
AR200iInt[76] := AR200iInterger76[iMainNo];
AR200iInt[77] := AR200iInterger77[iMainNo];
AR200iInt[78] := AR200iInterger78[iMainNo];
AR200iInt[79] := AR200iInterger79[iMainNo];
AR200iInt[80] := AR200iInterger80[iMainNo];
AR200iInt[81] := AR200iInterger81[iMainNo];
AR200iInt[82] := AR200iInterger82[iMainNo];
AR200iInt[83] := AR200iInterger83[iMainNo];
AR200iInt[84] := AR200iInterger84[iMainNo];
AR200iInt[85] := AR200iInterger85[iMainNo];
AR200iInt[86] := AR200iInterger86[iMainNo];
AR200iInt[87] := AR200iInterger87[iMainNo];
AR200iInt[88] := AR200iInterger88[iMainNo];
AR200iInt[89] := AR200iInterger89[iMainNo];
AR200iInt[90] := AR200iInterger90[iMainNo];
AR200iInt[91] := AR200iInterger91[iMainNo];
AR200iInt[92] := AR200iInterger92[iMainNo];
AR200iInt[93] := AR200iInterger93[iMainNo];
AR200iInt[94] := AR200iInterger94[iMainNo];
AR200iInt[95] := AR200iInterger95[iMainNo];
AR200iInt[96] := AR200iInterger96[iMainNo];
AR200iInt[97] := AR200iInterger97[iMainNo];
AR200iInt[98] := AR200iInterger98[iMainNo];
AR200iInt[99] := AR200iInterger99[iMainNo];
AR200iInt[100] := AR200iInterger100[iMainNo];




iSequencePresentProgram1 := AR200iInterger101[iMainNo];
iSequencePresentProgram2 := AR200iInterger102[iMainNo];
iSequencePresentProgram3 := AR200iInterger103[iMainNo];
iSequencePresentProgram4 := AR200iInterger104[iMainNo];
iSequencePresentProgram5 := AR200iInterger105[iMainNo];
iSequencePresentProgram6 := AR200iInterger106[iMainNo];
iSequencePresentProgram7 := AR200iInterger107[iMainNo];
iSequencePresentProgram8 := AR200iInterger108[iMainNo];
iSequencePresentProgram9 := AR200iInterger109[iMainNo];
iSequencePresentProgram10 := AR200iInterger110[iMainNo];



iSubProAdd1 := AR200iInt[((iSubNo*10)+1)-10];
iSubProAdd2 := AR200iInt[((iSubNo*10)+2)-10];
iSubProAdd3 := AR200iInt[((iSubNo*10)+3)-10];
iSubProAdd4 := AR200iInt[((iSubNo*10)+4)-10];
iSubProAdd5 := AR200iInt[((iSubNo*10)+5)-10];
iSubProAdd6 := AR200iInt[((iSubNo*10)+6)-10];
iSubProAdd7 := AR200iInt[((iSubNo*10)+7)-10];
iSubProAdd8 := AR200iInt[((iSubNo*10)+8)-10];
iSubProAdd9 := AR200iInt[((iSubNo*10)+9)-10];
iSubProAdd10 := AR200iInt[((iSubNo*10)+10)-10];




END_IF

SaveDF(CLK:=bSavePB,Q=>);

IF SaveDF.Q AND iMainNo>0 THEN

AR200iInt[((iSubNo*10)+1)-10] := iSubProAdd1;
AR200iInt[((iSubNo*10)+2)-10] := iSubProAdd2;
AR200iInt[((iSubNo*10)+3)-10] := iSubProAdd3;
AR200iInt[((iSubNo*10)+4)-10] := iSubProAdd4;
AR200iInt[((iSubNo*10)+5)-10] := iSubProAdd5;
AR200iInt[((iSubNo*10)+6)-10] := iSubProAdd6;
AR200iInt[((iSubNo*10)+7)-10] := iSubProAdd7;
AR200iInt[((iSubNo*10)+8)-10] := iSubProAdd8;
AR200iInt[((iSubNo*10)+9)-10] := iSubProAdd9;
AR200iInt[((iSubNo*10)+10)-10] := iSubProAdd10;



AR200iInterger1[iMainNo] := AR200iInt[1];
AR200iInterger2[iMainNo] := AR200iInt[2];
AR200iInterger3[iMainNo] := AR200iInt[3];
AR200iInterger4[iMainNo] := AR200iInt[4];
AR200iInterger5[iMainNo] := AR200iInt[5];
AR200iInterger6[iMainNo] := AR200iInt[6];
AR200iInterger7[iMainNo] := AR200iInt[7];
AR200iInterger8[iMainNo] := AR200iInt[8];
AR200iInterger9[iMainNo] := AR200iInt[9];
AR200iInterger10[iMainNo] := AR200iInt[10];
AR200iInterger11[iMainNo] := AR200iInt[11];
AR200iInterger12[iMainNo] := AR200iInt[12];
AR200iInterger13[iMainNo] := AR200iInt[13];
AR200iInterger14[iMainNo] := AR200iInt[14];
AR200iInterger15[iMainNo] := AR200iInt[15];
AR200iInterger16[iMainNo] := AR200iInt[16];
AR200iInterger17[iMainNo] := AR200iInt[17];
AR200iInterger18[iMainNo] := AR200iInt[18];
AR200iInterger19[iMainNo] := AR200iInt[19];
AR200iInterger20[iMainNo] := AR200iInt[20];
AR200iInterger21[iMainNo] := AR200iInt[21];
AR200iInterger22[iMainNo] := AR200iInt[22];
AR200iInterger23[iMainNo] := AR200iInt[23];
AR200iInterger24[iMainNo] := AR200iInt[24];
AR200iInterger25[iMainNo] := AR200iInt[25];
AR200iInterger26[iMainNo] := AR200iInt[26];
AR200iInterger27[iMainNo] := AR200iInt[27];
AR200iInterger28[iMainNo] := AR200iInt[28];
AR200iInterger29[iMainNo] := AR200iInt[29];
AR200iInterger30[iMainNo] := AR200iInt[30];
AR200iInterger31[iMainNo] := AR200iInt[31];
AR200iInterger32[iMainNo] := AR200iInt[32];
AR200iInterger33[iMainNo] := AR200iInt[33];
AR200iInterger34[iMainNo] := AR200iInt[34];
AR200iInterger35[iMainNo] := AR200iInt[35];
AR200iInterger36[iMainNo] := AR200iInt[36];
AR200iInterger37[iMainNo] := AR200iInt[37];
AR200iInterger38[iMainNo] := AR200iInt[38];
AR200iInterger39[iMainNo] := AR200iInt[39];
AR200iInterger40[iMainNo] := AR200iInt[40];
AR200iInterger41[iMainNo] := AR200iInt[41];
AR200iInterger42[iMainNo] := AR200iInt[42];
AR200iInterger43[iMainNo] := AR200iInt[43];
AR200iInterger44[iMainNo] := AR200iInt[44];
AR200iInterger45[iMainNo] := AR200iInt[45];
AR200iInterger46[iMainNo] := AR200iInt[46];
AR200iInterger47[iMainNo] := AR200iInt[47];
AR200iInterger48[iMainNo] := AR200iInt[48];
AR200iInterger49[iMainNo] := AR200iInt[49];
AR200iInterger50[iMainNo] := AR200iInt[50];
AR200iInterger51[iMainNo] := AR200iInt[51];
AR200iInterger52[iMainNo] := AR200iInt[52];
AR200iInterger53[iMainNo] := AR200iInt[53];
AR200iInterger54[iMainNo] := AR200iInt[54];
AR200iInterger55[iMainNo] := AR200iInt[55];
AR200iInterger56[iMainNo] := AR200iInt[56];
AR200iInterger57[iMainNo] := AR200iInt[57];
AR200iInterger58[iMainNo] := AR200iInt[58];
AR200iInterger59[iMainNo] := AR200iInt[59];
AR200iInterger60[iMainNo] := AR200iInt[60];
AR200iInterger61[iMainNo] := AR200iInt[61];
AR200iInterger62[iMainNo] := AR200iInt[62];
AR200iInterger63[iMainNo] := AR200iInt[63];
AR200iInterger64[iMainNo] := AR200iInt[64];
AR200iInterger65[iMainNo] := AR200iInt[65];
AR200iInterger66[iMainNo] := AR200iInt[66];
AR200iInterger67[iMainNo] := AR200iInt[67];
AR200iInterger68[iMainNo] := AR200iInt[68];
AR200iInterger69[iMainNo] := AR200iInt[69];
AR200iInterger70[iMainNo] := AR200iInt[70];
AR200iInterger71[iMainNo] := AR200iInt[71];
AR200iInterger72[iMainNo] := AR200iInt[72];
AR200iInterger73[iMainNo] := AR200iInt[73];
AR200iInterger74[iMainNo] := AR200iInt[74];
AR200iInterger75[iMainNo] := AR200iInt[75];
AR200iInterger76[iMainNo] := AR200iInt[76];
AR200iInterger77[iMainNo] := AR200iInt[77];
AR200iInterger78[iMainNo] := AR200iInt[78];
AR200iInterger79[iMainNo] := AR200iInt[79];
AR200iInterger80[iMainNo] := AR200iInt[80];
AR200iInterger81[iMainNo] := AR200iInt[81];
AR200iInterger82[iMainNo] := AR200iInt[82];
AR200iInterger83[iMainNo] := AR200iInt[83];
AR200iInterger84[iMainNo] := AR200iInt[84];
AR200iInterger85[iMainNo] := AR200iInt[85];
AR200iInterger86[iMainNo] := AR200iInt[86];
AR200iInterger87[iMainNo] := AR200iInt[87];
AR200iInterger88[iMainNo] := AR200iInt[88];
AR200iInterger89[iMainNo] := AR200iInt[89];
AR200iInterger90[iMainNo] := AR200iInt[90];
AR200iInterger91[iMainNo] := AR200iInt[91];
AR200iInterger92[iMainNo] := AR200iInt[92];
AR200iInterger93[iMainNo] := AR200iInt[93];
AR200iInterger94[iMainNo] := AR200iInt[94];
AR200iInterger95[iMainNo] := AR200iInt[95];
AR200iInterger96[iMainNo] := AR200iInt[96];
AR200iInterger97[iMainNo] := AR200iInt[97];
AR200iInterger98[iMainNo] := AR200iInt[98];
AR200iInterger99[iMainNo] := AR200iInt[99];
AR200iInterger100[iMainNo] := AR200iInt[100];

AR200iInterger101[iMainNo] := iSequencePresentProgram1;
AR200iInterger102[iMainNo] := iSequencePresentProgram2;
AR200iInterger103[iMainNo] := iSequencePresentProgram3;
AR200iInterger104[iMainNo] := iSequencePresentProgram4;
AR200iInterger105[iMainNo] := iSequencePresentProgram5;
AR200iInterger106[iMainNo] := iSequencePresentProgram6;
AR200iInterger107[iMainNo] := iSequencePresentProgram7;
AR200iInterger108[iMainNo] := iSequencePresentProgram8;
AR200iInterger109[iMainNo] := iSequencePresentProgram9;
AR200iInterger110[iMainNo] := iSequencePresentProgram10;


END_IF


(*Call Recipe*)


IF iCallMainRecipeNo>0 AND iCallMainRecipeNo<100 OR iCallSubRecipeNo>0 AND iCallSubRecipeNo<11 THEN

AR200iIntCall[1] := AR200iInterger1[iCallMainRecipeNo];
AR200iIntCall[2] := AR200iInterger2[iCallMainRecipeNo];
AR200iIntCall[3] := AR200iInterger3[iCallMainRecipeNo];
AR200iIntCall[4] := AR200iInterger4[iCallMainRecipeNo];
AR200iIntCall[5] := AR200iInterger5[iCallMainRecipeNo];
AR200iIntCall[6] := AR200iInterger6[iCallMainRecipeNo];
AR200iIntCall[7] := AR200iInterger7[iCallMainRecipeNo];
AR200iIntCall[8] := AR200iInterger8[iCallMainRecipeNo];
AR200iIntCall[9] := AR200iInterger9[iCallMainRecipeNo];
AR200iIntCall[10] := AR200iInterger10[iCallMainRecipeNo];
AR200iIntCall[11] := AR200iInterger11[iCallMainRecipeNo];
AR200iIntCall[12] := AR200iInterger12[iCallMainRecipeNo];
AR200iIntCall[13] := AR200iInterger13[iCallMainRecipeNo];
AR200iIntCall[14] := AR200iInterger14[iCallMainRecipeNo];
AR200iIntCall[15] := AR200iInterger15[iCallMainRecipeNo];
AR200iIntCall[16] := AR200iInterger16[iCallMainRecipeNo];
AR200iIntCall[17] := AR200iInterger17[iCallMainRecipeNo];
AR200iIntCall[18] := AR200iInterger18[iCallMainRecipeNo];
AR200iIntCall[19] := AR200iInterger19[iCallMainRecipeNo];
AR200iIntCall[20] := AR200iInterger20[iCallMainRecipeNo];
AR200iIntCall[21] := AR200iInterger21[iCallMainRecipeNo];
AR200iIntCall[22] := AR200iInterger22[iCallMainRecipeNo];
AR200iIntCall[23] := AR200iInterger23[iCallMainRecipeNo];
AR200iIntCall[24] := AR200iInterger24[iCallMainRecipeNo];
AR200iIntCall[25] := AR200iInterger25[iCallMainRecipeNo];
AR200iIntCall[26] := AR200iInterger26[iCallMainRecipeNo];
AR200iIntCall[27] := AR200iInterger27[iCallMainRecipeNo];
AR200iIntCall[28] := AR200iInterger28[iCallMainRecipeNo];
AR200iIntCall[29] := AR200iInterger29[iCallMainRecipeNo];
AR200iIntCall[30] := AR200iInterger30[iCallMainRecipeNo];
AR200iIntCall[31] := AR200iInterger31[iCallMainRecipeNo];
AR200iIntCall[32] := AR200iInterger32[iCallMainRecipeNo];
AR200iIntCall[33] := AR200iInterger33[iCallMainRecipeNo];
AR200iIntCall[34] := AR200iInterger34[iCallMainRecipeNo];
AR200iIntCall[35] := AR200iInterger35[iCallMainRecipeNo];
AR200iIntCall[36] := AR200iInterger36[iCallMainRecipeNo];
AR200iIntCall[37] := AR200iInterger37[iCallMainRecipeNo];
AR200iIntCall[38] := AR200iInterger38[iCallMainRecipeNo];
AR200iIntCall[39] := AR200iInterger39[iCallMainRecipeNo];
AR200iIntCall[40] := AR200iInterger40[iCallMainRecipeNo];
AR200iIntCall[41] := AR200iInterger41[iCallMainRecipeNo];
AR200iIntCall[42] := AR200iInterger42[iCallMainRecipeNo];
AR200iIntCall[43] := AR200iInterger43[iCallMainRecipeNo];
AR200iIntCall[44] := AR200iInterger44[iCallMainRecipeNo];
AR200iIntCall[45] := AR200iInterger45[iCallMainRecipeNo];
AR200iIntCall[46] := AR200iInterger46[iCallMainRecipeNo];
AR200iIntCall[47] := AR200iInterger47[iCallMainRecipeNo];
AR200iIntCall[48] := AR200iInterger48[iCallMainRecipeNo];
AR200iIntCall[49] := AR200iInterger49[iCallMainRecipeNo];
AR200iIntCall[50] := AR200iInterger50[iCallMainRecipeNo];
AR200iIntCall[51] := AR200iInterger51[iCallMainRecipeNo];
AR200iIntCall[52] := AR200iInterger52[iCallMainRecipeNo];
AR200iIntCall[53] := AR200iInterger53[iCallMainRecipeNo];
AR200iIntCall[54] := AR200iInterger54[iCallMainRecipeNo];
AR200iIntCall[55] := AR200iInterger55[iCallMainRecipeNo];
AR200iIntCall[56] := AR200iInterger56[iCallMainRecipeNo];
AR200iIntCall[57] := AR200iInterger57[iCallMainRecipeNo];
AR200iIntCall[58] := AR200iInterger58[iCallMainRecipeNo];
AR200iIntCall[59] := AR200iInterger59[iCallMainRecipeNo];
AR200iIntCall[60] := AR200iInterger60[iCallMainRecipeNo];
AR200iIntCall[61] := AR200iInterger61[iCallMainRecipeNo];
AR200iIntCall[62] := AR200iInterger62[iCallMainRecipeNo];
AR200iIntCall[63] := AR200iInterger63[iCallMainRecipeNo];
AR200iIntCall[64] := AR200iInterger64[iCallMainRecipeNo];
AR200iIntCall[65] := AR200iInterger65[iCallMainRecipeNo];
AR200iIntCall[66] := AR200iInterger66[iCallMainRecipeNo];
AR200iIntCall[67] := AR200iInterger67[iCallMainRecipeNo];
AR200iIntCall[68] := AR200iInterger68[iCallMainRecipeNo];
AR200iIntCall[69] := AR200iInterger69[iCallMainRecipeNo];
AR200iIntCall[70] := AR200iInterger70[iCallMainRecipeNo];
AR200iIntCall[71] := AR200iInterger71[iCallMainRecipeNo];
AR200iIntCall[72] := AR200iInterger72[iCallMainRecipeNo];
AR200iIntCall[73] := AR200iInterger73[iCallMainRecipeNo];
AR200iIntCall[74] := AR200iInterger74[iCallMainRecipeNo];
AR200iIntCall[75] := AR200iInterger75[iCallMainRecipeNo];
AR200iIntCall[76] := AR200iInterger76[iCallMainRecipeNo];
AR200iIntCall[77] := AR200iInterger77[iCallMainRecipeNo];
AR200iIntCall[78] := AR200iInterger78[iCallMainRecipeNo];
AR200iIntCall[79] := AR200iInterger79[iCallMainRecipeNo];
AR200iIntCall[80] := AR200iInterger80[iCallMainRecipeNo];
AR200iIntCall[81] := AR200iInterger81[iCallMainRecipeNo];
AR200iIntCall[82] := AR200iInterger82[iCallMainRecipeNo];
AR200iIntCall[83] := AR200iInterger83[iCallMainRecipeNo];
AR200iIntCall[84] := AR200iInterger84[iCallMainRecipeNo];
AR200iIntCall[85] := AR200iInterger85[iCallMainRecipeNo];
AR200iIntCall[86] := AR200iInterger86[iCallMainRecipeNo];
AR200iIntCall[87] := AR200iInterger87[iCallMainRecipeNo];
AR200iIntCall[88] := AR200iInterger88[iCallMainRecipeNo];
AR200iIntCall[89] := AR200iInterger89[iCallMainRecipeNo];
AR200iIntCall[90] := AR200iInterger90[iCallMainRecipeNo];
AR200iIntCall[91] := AR200iInterger91[iCallMainRecipeNo];
AR200iIntCall[92] := AR200iInterger92[iCallMainRecipeNo];
AR200iIntCall[93] := AR200iInterger93[iCallMainRecipeNo];
AR200iIntCall[94] := AR200iInterger94[iCallMainRecipeNo];
AR200iIntCall[95] := AR200iInterger95[iCallMainRecipeNo];
AR200iIntCall[96] := AR200iInterger96[iCallMainRecipeNo];
AR200iIntCall[97] := AR200iInterger97[iCallMainRecipeNo];
AR200iIntCall[98] := AR200iInterger98[iCallMainRecipeNo];
AR200iIntCall[99] := AR200iInterger99[iCallMainRecipeNo];
AR200iIntCall[100] := AR200iInterger100[iCallMainRecipeNo];

END_IF


IF iCallMainRecipeNo>0 AND iCallMainRecipeNo<100  THEN

iSeqCallPresentProgram1 := AR200iInterger101[iCallMainRecipeNo];
iSeqCallPresentProgram2 := AR200iInterger102[iCallMainRecipeNo];
iSeqCallPresentProgram3 := AR200iInterger103[iCallMainRecipeNo];
iSeqCallPresentProgram4 := AR200iInterger104[iCallMainRecipeNo];
iSeqCallPresentProgram5 := AR200iInterger105[iCallMainRecipeNo];
iSeqCallPresentProgram6 := AR200iInterger106[iCallMainRecipeNo];
iSeqCallPresentProgram7 := AR200iInterger107[iCallMainRecipeNo];
iSeqCallPresentProgram8 := AR200iInterger108[iCallMainRecipeNo];
iSeqCallPresentProgram9 := AR200iInterger109[iCallMainRecipeNo];
iSeqCallPresentProgram10 := AR200iInterger110[iCallMainRecipeNo];
END_IF


IF  iCallSubRecipeNo>0 AND iCallSubRecipeNo<11 THEN

iCallSubProAdd1 :=AR200iIntCall[((iCallSubRecipeNo*10)+1)-10];
iCallSubProAdd2 :=AR200iIntCall[((iCallSubRecipeNo*10)+2)-10];
iCallSubProAdd3 :=AR200iIntCall[((iCallSubRecipeNo*10)+3)-10];
iCallSubProAdd4 :=AR200iIntCall[((iCallSubRecipeNo*10)+4)-10];
iCallSubProAdd5 :=AR200iIntCall[((iCallSubRecipeNo*10)+5)-10];
iCallSubProAdd6 :=AR200iIntCall[((iCallSubRecipeNo*10)+6)-10];
iCallSubProAdd7 :=AR200iIntCall[((iCallSubRecipeNo*10)+7)-10];
iCallSubProAdd8 :=AR200iIntCall[((iCallSubRecipeNo*10)+8)-10];
iCallSubProAdd9 :=AR200iIntCall[((iCallSubRecipeNo*10)+9)-10];
iCallSubProAdd10 :=AR200iIntCall[((iCallSubRecipeNo*10)+10)-10];
END_IF

IF iCallMainRecipeNo<=0 OR iCallMainRecipeNo >=100 THEN


iSeqCallPresentProgram1 := 0;
iSeqCallPresentProgram2 := 0;
iSeqCallPresentProgram3 := 0;
iSeqCallPresentProgram4 := 0;
iSeqCallPresentProgram5 := 0;
iSeqCallPresentProgram6 := 0;
iSeqCallPresentProgram7 := 0;
iSeqCallPresentProgram8 := 0;
iSeqCallPresentProgram9 := 0;
iSeqCallPresentProgram10 := 0;
END_IF


IF iCallMainRecipeNo>=100 OR iCallMainRecipeNo<=0 OR iCallSubRecipeNo>=11 OR iCallSubRecipeNo<=0 THEN

iCallSubProAdd1 :=0;
iCallSubProAdd2 :=0;
iCallSubProAdd3 :=0;
iCallSubProAdd4 :=0;
iCallSubProAdd5 :=0;
iCallSubProAdd6 :=0;
iCallSubProAdd7 :=0;
iCallSubProAdd8 :=0;
iCallSubProAdd9 :=0;
iCallSubProAdd10 :=0;
END_IF



(*Scan Total Time*)


IF iTotalTimeMainRecipeNo >0 OR iTotalTimeSubRecipeNo > 0 THEN

AR200iTotalTimeIntCall[1] := AR200iInterger1[iTotalTimeMainRecipeNo];
AR200iTotalTimeIntCall[2] := AR200iInterger2[iTotalTimeMainRecipeNo];
AR200iTotalTimeIntCall[3] := AR200iInterger3[iTotalTimeMainRecipeNo];
AR200iTotalTimeIntCall[4] := AR200iInterger4[iTotalTimeMainRecipeNo];
AR200iTotalTimeIntCall[5] := AR200iInterger5[iTotalTimeMainRecipeNo];
AR200iTotalTimeIntCall[6] := AR200iInterger6[iTotalTimeMainRecipeNo];
AR200iTotalTimeIntCall[7] := AR200iInterger7[iTotalTimeMainRecipeNo];
AR200iTotalTimeIntCall[8] := AR200iInterger8[iTotalTimeMainRecipeNo];
AR200iTotalTimeIntCall[9] := AR200iInterger9[iTotalTimeMainRecipeNo];
AR200iTotalTimeIntCall[10] := AR200iInterger10[iTotalTimeMainRecipeNo];
AR200iTotalTimeIntCall[11] := AR200iInterger11[iTotalTimeMainRecipeNo];
AR200iTotalTimeIntCall[12] := AR200iInterger12[iTotalTimeMainRecipeNo];
AR200iTotalTimeIntCall[13] := AR200iInterger13[iTotalTimeMainRecipeNo];
AR200iTotalTimeIntCall[14] := AR200iInterger14[iTotalTimeMainRecipeNo];
AR200iTotalTimeIntCall[15] := AR200iInterger15[iTotalTimeMainRecipeNo];
AR200iTotalTimeIntCall[16] := AR200iInterger16[iTotalTimeMainRecipeNo];
AR200iTotalTimeIntCall[17] := AR200iInterger17[iTotalTimeMainRecipeNo];
AR200iTotalTimeIntCall[18] := AR200iInterger18[iTotalTimeMainRecipeNo];
AR200iTotalTimeIntCall[19] := AR200iInterger19[iTotalTimeMainRecipeNo];
AR200iTotalTimeIntCall[20] := AR200iInterger20[iTotalTimeMainRecipeNo];
AR200iTotalTimeIntCall[21] := AR200iInterger21[iTotalTimeMainRecipeNo];
AR200iTotalTimeIntCall[22] := AR200iInterger22[iTotalTimeMainRecipeNo];
AR200iTotalTimeIntCall[23] := AR200iInterger23[iTotalTimeMainRecipeNo];
AR200iTotalTimeIntCall[24] := AR200iInterger24[iTotalTimeMainRecipeNo];
AR200iTotalTimeIntCall[25] := AR200iInterger25[iTotalTimeMainRecipeNo];
AR200iTotalTimeIntCall[26] := AR200iInterger26[iTotalTimeMainRecipeNo];
AR200iTotalTimeIntCall[27] := AR200iInterger27[iTotalTimeMainRecipeNo];
AR200iTotalTimeIntCall[28] := AR200iInterger28[iTotalTimeMainRecipeNo];
AR200iTotalTimeIntCall[29] := AR200iInterger29[iTotalTimeMainRecipeNo];
AR200iTotalTimeIntCall[30] := AR200iInterger30[iTotalTimeMainRecipeNo];
AR200iTotalTimeIntCall[31] := AR200iInterger31[iTotalTimeMainRecipeNo];
AR200iTotalTimeIntCall[32] := AR200iInterger32[iTotalTimeMainRecipeNo];
AR200iTotalTimeIntCall[33] := AR200iInterger33[iTotalTimeMainRecipeNo];
AR200iTotalTimeIntCall[34] := AR200iInterger34[iTotalTimeMainRecipeNo];
AR200iTotalTimeIntCall[35] := AR200iInterger35[iTotalTimeMainRecipeNo];
AR200iTotalTimeIntCall[36] := AR200iInterger36[iTotalTimeMainRecipeNo];
AR200iTotalTimeIntCall[37] := AR200iInterger37[iTotalTimeMainRecipeNo];
AR200iTotalTimeIntCall[38] := AR200iInterger38[iTotalTimeMainRecipeNo];
AR200iTotalTimeIntCall[39] := AR200iInterger39[iTotalTimeMainRecipeNo];
AR200iTotalTimeIntCall[40] := AR200iInterger40[iTotalTimeMainRecipeNo];
AR200iTotalTimeIntCall[41] := AR200iInterger41[iTotalTimeMainRecipeNo];
AR200iTotalTimeIntCall[42] := AR200iInterger42[iTotalTimeMainRecipeNo];
AR200iTotalTimeIntCall[43] := AR200iInterger43[iTotalTimeMainRecipeNo];
AR200iTotalTimeIntCall[44] := AR200iInterger44[iTotalTimeMainRecipeNo];
AR200iTotalTimeIntCall[45] := AR200iInterger45[iTotalTimeMainRecipeNo];
AR200iTotalTimeIntCall[46] := AR200iInterger46[iTotalTimeMainRecipeNo];
AR200iTotalTimeIntCall[47] := AR200iInterger47[iTotalTimeMainRecipeNo];
AR200iTotalTimeIntCall[48] := AR200iInterger48[iTotalTimeMainRecipeNo];
AR200iTotalTimeIntCall[49] := AR200iInterger49[iTotalTimeMainRecipeNo];
AR200iTotalTimeIntCall[50] := AR200iInterger50[iTotalTimeMainRecipeNo];
AR200iTotalTimeIntCall[51] := AR200iInterger51[iTotalTimeMainRecipeNo];
AR200iTotalTimeIntCall[52] := AR200iInterger52[iTotalTimeMainRecipeNo];
AR200iTotalTimeIntCall[53] := AR200iInterger53[iTotalTimeMainRecipeNo];
AR200iTotalTimeIntCall[54] := AR200iInterger54[iTotalTimeMainRecipeNo];
AR200iTotalTimeIntCall[55] := AR200iInterger55[iTotalTimeMainRecipeNo];
AR200iTotalTimeIntCall[56] := AR200iInterger56[iTotalTimeMainRecipeNo];
AR200iTotalTimeIntCall[57] := AR200iInterger57[iTotalTimeMainRecipeNo];
AR200iTotalTimeIntCall[58] := AR200iInterger58[iTotalTimeMainRecipeNo];
AR200iTotalTimeIntCall[59] := AR200iInterger59[iTotalTimeMainRecipeNo];
AR200iTotalTimeIntCall[60] := AR200iInterger60[iTotalTimeMainRecipeNo];
AR200iTotalTimeIntCall[61] := AR200iInterger61[iTotalTimeMainRecipeNo];
AR200iTotalTimeIntCall[62] := AR200iInterger62[iTotalTimeMainRecipeNo];
AR200iTotalTimeIntCall[63] := AR200iInterger63[iTotalTimeMainRecipeNo];
AR200iTotalTimeIntCall[64] := AR200iInterger64[iTotalTimeMainRecipeNo];
AR200iTotalTimeIntCall[65] := AR200iInterger65[iTotalTimeMainRecipeNo];
AR200iTotalTimeIntCall[66] := AR200iInterger66[iTotalTimeMainRecipeNo];
AR200iTotalTimeIntCall[67] := AR200iInterger67[iTotalTimeMainRecipeNo];
AR200iTotalTimeIntCall[68] := AR200iInterger68[iTotalTimeMainRecipeNo];
AR200iTotalTimeIntCall[69] := AR200iInterger69[iTotalTimeMainRecipeNo];
AR200iTotalTimeIntCall[70] := AR200iInterger70[iTotalTimeMainRecipeNo];
AR200iTotalTimeIntCall[71] := AR200iInterger71[iTotalTimeMainRecipeNo];
AR200iTotalTimeIntCall[72] := AR200iInterger72[iTotalTimeMainRecipeNo];
AR200iTotalTimeIntCall[73] := AR200iInterger73[iTotalTimeMainRecipeNo];
AR200iTotalTimeIntCall[74] := AR200iInterger74[iTotalTimeMainRecipeNo];
AR200iTotalTimeIntCall[75] := AR200iInterger75[iTotalTimeMainRecipeNo];
AR200iTotalTimeIntCall[76] := AR200iInterger76[iTotalTimeMainRecipeNo];
AR200iTotalTimeIntCall[77] := AR200iInterger77[iTotalTimeMainRecipeNo];
AR200iTotalTimeIntCall[78] := AR200iInterger78[iTotalTimeMainRecipeNo];
AR200iTotalTimeIntCall[79] := AR200iInterger79[iTotalTimeMainRecipeNo];
AR200iTotalTimeIntCall[80] := AR200iInterger80[iTotalTimeMainRecipeNo];
AR200iTotalTimeIntCall[81] := AR200iInterger81[iTotalTimeMainRecipeNo];
AR200iTotalTimeIntCall[82] := AR200iInterger82[iTotalTimeMainRecipeNo];
AR200iTotalTimeIntCall[83] := AR200iInterger83[iTotalTimeMainRecipeNo];
AR200iTotalTimeIntCall[84] := AR200iInterger84[iTotalTimeMainRecipeNo];
AR200iTotalTimeIntCall[85] := AR200iInterger85[iTotalTimeMainRecipeNo];
AR200iTotalTimeIntCall[86] := AR200iInterger86[iTotalTimeMainRecipeNo];
AR200iTotalTimeIntCall[87] := AR200iInterger87[iTotalTimeMainRecipeNo];
AR200iTotalTimeIntCall[88] := AR200iInterger88[iTotalTimeMainRecipeNo];
AR200iTotalTimeIntCall[89] := AR200iInterger89[iTotalTimeMainRecipeNo];
AR200iTotalTimeIntCall[90] := AR200iInterger90[iTotalTimeMainRecipeNo];
AR200iTotalTimeIntCall[91] := AR200iInterger91[iTotalTimeMainRecipeNo];
AR200iTotalTimeIntCall[92] := AR200iInterger92[iTotalTimeMainRecipeNo];
AR200iTotalTimeIntCall[93] := AR200iInterger93[iTotalTimeMainRecipeNo];
AR200iTotalTimeIntCall[94] := AR200iInterger94[iTotalTimeMainRecipeNo];
AR200iTotalTimeIntCall[95] := AR200iInterger95[iTotalTimeMainRecipeNo];
AR200iTotalTimeIntCall[96] := AR200iInterger96[iTotalTimeMainRecipeNo];
AR200iTotalTimeIntCall[97] := AR200iInterger97[iTotalTimeMainRecipeNo];
AR200iTotalTimeIntCall[98] := AR200iInterger98[iTotalTimeMainRecipeNo];
AR200iTotalTimeIntCall[99] := AR200iInterger99[iTotalTimeMainRecipeNo];
AR200iTotalTimeIntCall[100] := AR200iInterger100[iTotalTimeMainRecipeNo];


		IF  iTotalTimeMainRecipeNo >0 AND  iCallRecipeTotalTime = 0THEN


		iSeqCallTTPresentProgram1 := AR200iInterger101[iTotalTimeMainRecipeNo];
		iSeqCallTTPresentProgram2 := AR200iInterger102[iTotalTimeMainRecipeNo];
		iSeqCallTTPresentProgram3 := AR200iInterger103[iTotalTimeMainRecipeNo];
		iSeqCallTTPresentProgram4 := AR200iInterger104[iTotalTimeMainRecipeNo];
		iSeqCallTTPresentProgram5 := AR200iInterger105[iTotalTimeMainRecipeNo];
		iSeqCallTTPresentProgram6 := AR200iInterger106[iTotalTimeMainRecipeNo];
		iSeqCallTTPresentProgram7 := AR200iInterger107[iTotalTimeMainRecipeNo];
		iSeqCallTTPresentProgram8 := AR200iInterger108[iTotalTimeMainRecipeNo];
		iSeqCallTTPresentProgram9 := AR200iInterger109[iTotalTimeMainRecipeNo];
		iSeqCallTTPresentProgram10 := AR200iInterger110[iTotalTimeMainRecipeNo];
	

		iCallRecipeTotalTime :=
		AR200iTotalTimeIntCall[((iSeqCallTTPresentProgram1*10)+1)-10] +
		AR200iTotalTimeIntCall[((iSeqCallTTPresentProgram2*10)+1)-10] +
		AR200iTotalTimeIntCall[((iSeqCallTTPresentProgram3*10)+1)-10] +
		AR200iTotalTimeIntCall[((iSeqCallTTPresentProgram4*10)+1)-10] +
		AR200iTotalTimeIntCall[((iSeqCallTTPresentProgram5*10)+1)-10] +
		AR200iTotalTimeIntCall[((iSeqCallTTPresentProgram6*10)+1)-10] +
		AR200iTotalTimeIntCall[((iSeqCallTTPresentProgram7*10)+1)-10] +
		AR200iTotalTimeIntCall[((iSeqCallTTPresentProgram8*10)+1)-10] +
		AR200iTotalTimeIntCall[((iSeqCallTTPresentProgram9*10)+1)-10] +
		AR200iTotalTimeIntCall[((iSeqCallTTPresentProgram10*10)+1)-10] ;


		END_IF


		IF iTotalTimeSubRecipeNo > 0 THEN

		AR10_iCallSubProTotalTime[1] :=AR200iTotalTimeIntCall[((iTotalTimeSubRecipeNo*10)+1)-10];
		AR10_iCallSubProTotalTime[2] :=AR200iTotalTimeIntCall[((iTotalTimeSubRecipeNo*10)+2)-10];
		AR10_iCallSubProTotalTime[3] :=AR200iTotalTimeIntCall[((iTotalTimeSubRecipeNo*10)+3)-10];
		AR10_iCallSubProTotalTime[4] :=AR200iTotalTimeIntCall[((iTotalTimeSubRecipeNo*10)+4)-10];
		AR10_iCallSubProTotalTime[5] :=AR200iTotalTimeIntCall[((iTotalTimeSubRecipeNo*10)+5)-10];
		AR10_iCallSubProTotalTime[6] :=AR200iTotalTimeIntCall[((iTotalTimeSubRecipeNo*10)+6)-10];
		AR10_iCallSubProTotalTime[7] :=AR200iTotalTimeIntCall[((iTotalTimeSubRecipeNo*10)+7)-10];
		AR10_iCallSubProTotalTime[8] :=AR200iTotalTimeIntCall[((iTotalTimeSubRecipeNo*10)+8)-10];
		AR10_iCallSubProTotalTime[9] :=AR200iTotalTimeIntCall[((iTotalTimeSubRecipeNo*10)+9)-10];
		AR10_iCallSubProTotalTime[10] :=AR200iTotalTimeIntCall[((iTotalTimeSubRecipeNo*10)+10)-10];

		END_IF

END_IF




IF  iTotalTimeMainRecipeNo <=0 THEN
iCallRecipeTotalTime := 0;
END_IF

		IF iTotalTimeSubRecipeNo <=0 THEN

		AR10_iCallSubProTotalTime[1] :=0;
		AR10_iCallSubProTotalTime[2] :=0;
		AR10_iCallSubProTotalTime[3] :=0;
		AR10_iCallSubProTotalTime[4] :=0;
		AR10_iCallSubProTotalTime[5] :=0;
		AR10_iCallSubProTotalTime[6] :=0;
		AR10_iCallSubProTotalTime[7] :=0;
		AR10_iCallSubProTotalTime[8] :=0;
		AR10_iCallSubProTotalTime[9] :=0;
		AR10_iCallSubProTotalTime[10] :=0;

		END_IF

END_FUNCTION_BLOCK

// ---- FBs/B_JKS_CustomFB/Other/fbUld3ZoneConveyorCtrl.TcPOU
FUNCTION_BLOCK fbUld3ZoneConveyorCtrl
VAR_INPUT
	bEnable		: BOOL;
	bRapidPB	: BOOL;
	bZone1Sensor	: BOOL;
	bZone2Sensor	: BOOL;
	bEndZoneSensor	: BOOL;
	diZone1BasketConfirmDelayTime	: DINT;
	diZone2BasketConfirmDelayTime	: DINT;
	diEndZoneBasketConfirmDelayTime	: DINT;
	diRapidPBDelayTime	: DINT;

	bEmergencyStop: BOOL;
END_VAR
VAR_OUTPUT
	bMotorOnOff	: BOOL;
END_VAR
VAR
	TON1: TON;
	TRIG1: R_TRIG;
	bMotorStopBit: BOOL;
	TON2: TON;
	Trig2: R_TRIG;
	TON3: TON;
	RampIn: BOOL;
	TON4: TON;
	bConvAutoCut: BOOL;
	CVDelayOff : BOOL;
	TON5: TON;
END_VAR

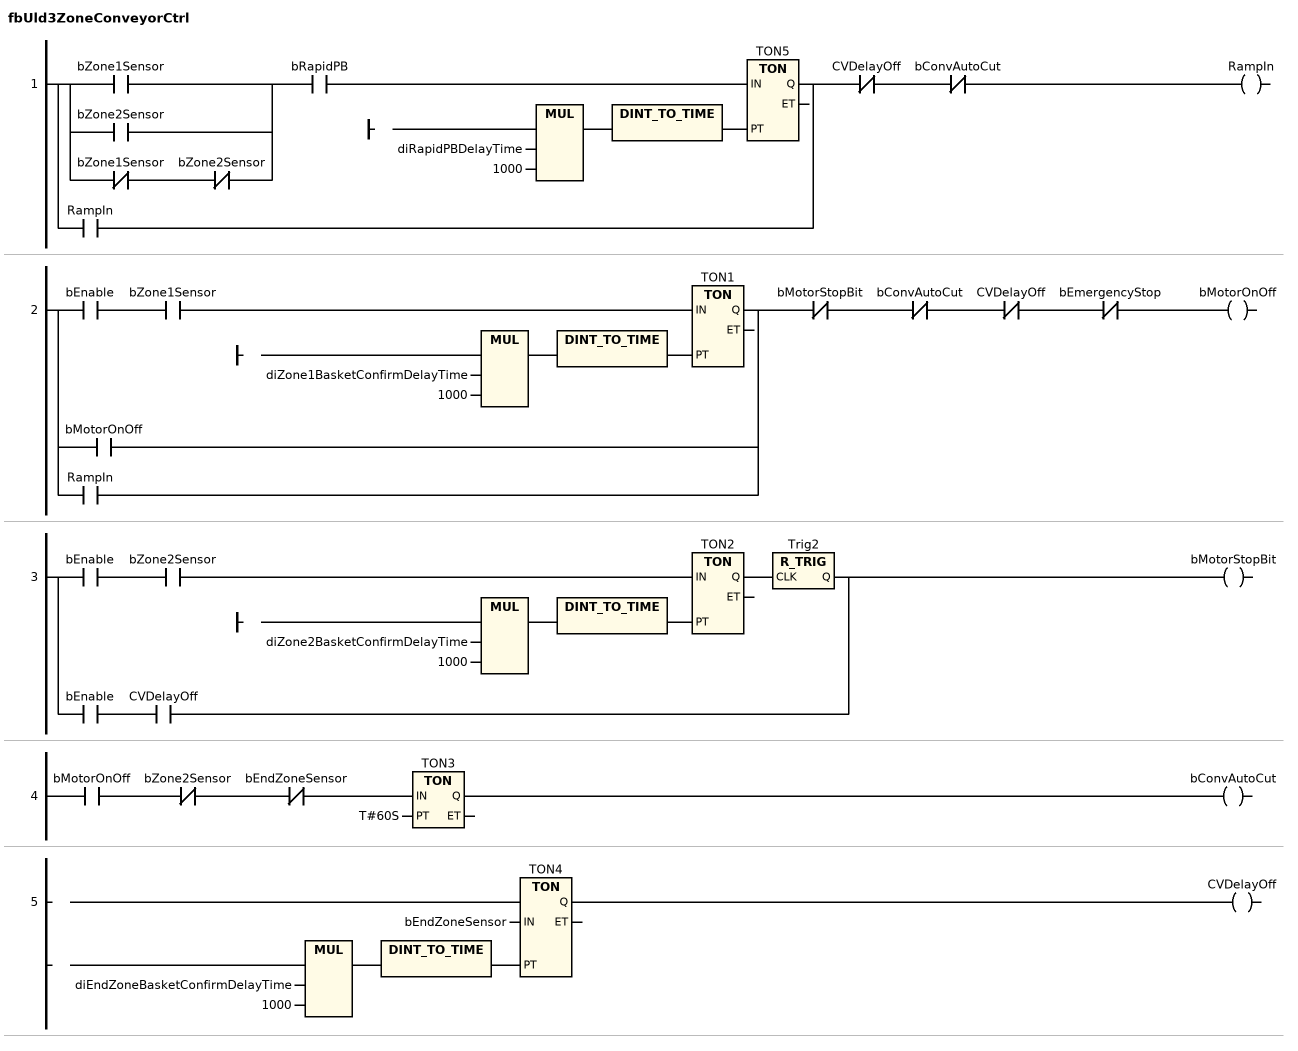
// NETWORK 1
TON5(IN := (bZone1Sensor OR bZone2Sensor OR NOT bZone1Sensor AND NOT bZone2Sensor) AND bRapidPB, PT := DINT_TO_TIME(diRapidPBDelayTime * 1000)); // TON
RampIn := (TON5.Q OR RampIn) AND NOT CVDelayOff AND NOT bConvAutoCut;

// NETWORK 2
TON1(IN := bEnable AND bZone1Sensor, PT := DINT_TO_TIME(diZone1BasketConfirmDelayTime * 1000)); // TON
bMotorOnOff := (TON1.Q OR bMotorOnOff OR RampIn) AND NOT bMotorStopBit AND NOT bConvAutoCut AND NOT CVDelayOff AND NOT bEmergencyStop;

// NETWORK 3
TON2(IN := bEnable AND bZone2Sensor, PT := DINT_TO_TIME(diZone2BasketConfirmDelayTime * 1000)); // TON
Trig2(CLK := TON2.Q); // R_TRIG
bMotorStopBit := Trig2.Q OR bEnable AND CVDelayOff;

// NETWORK 4
TON3(IN := bMotorOnOff AND NOT bZone2Sensor AND NOT bEndZoneSensor, PT := T#60S); // TON
bConvAutoCut := TON3.Q;

// NETWORK 5
TON4(IN := bEndZoneSensor, PT := DINT_TO_TIME(diEndZoneBasketConfirmDelayTime * 1000)); // TON
CVDelayOff := TON4.Q;

END_FUNCTION_BLOCK

// ---- FBs/B_JKS_CustomFB/Other/fbUldConveyor3Zones.TcPOU
FUNCTION_BLOCK fbUldConveyor3Zones
VAR_INPUT

	bEnable		: BOOL;
	bRapidPB	: BOOL;
	bUldBasketZone1TransferMemoryBit: BOOL;
	bUldBasketZone1ConfirmMemoryBit: BOOL;
	bUldBasketZone2TransferMemoryBit: BOOL;
	bUldBasketZone2ConfirmMemoryBit	: BOOL;

	bUldSensor1: BOOL;
	bUldSensor2: BOOL;
	bUldEndSensor: BOOL;
(*
	diZone1BasketConfirmDelayTime	: DINT;
	diZone2BasketConfirmDelayTime	: DINT;
	diRapidPBDelayTime	: DINT;
*)
	diEndZoneBasketConfirmDelayTime	: DINT;

	bEmergencyStop: BOOL;
END_VAR
VAR_OUTPUT
	bMotorOnOff	: BOOL;
END_VAR
VAR
	bRapidPBRE: R_TRIG;
	bMotorStopBit: BOOL;
	TON1: TON;
	TON2: TON;
	bConvAutoCut: BOOL;

	(*TRIG1: R_TRIG;
	Trig2: R_TRIG;
	TON3: TON;
	RampIn: BOOL;
	TON4: TON;
	CVDelayOff : BOOL;
	TON5: TON;*)

END_VAR

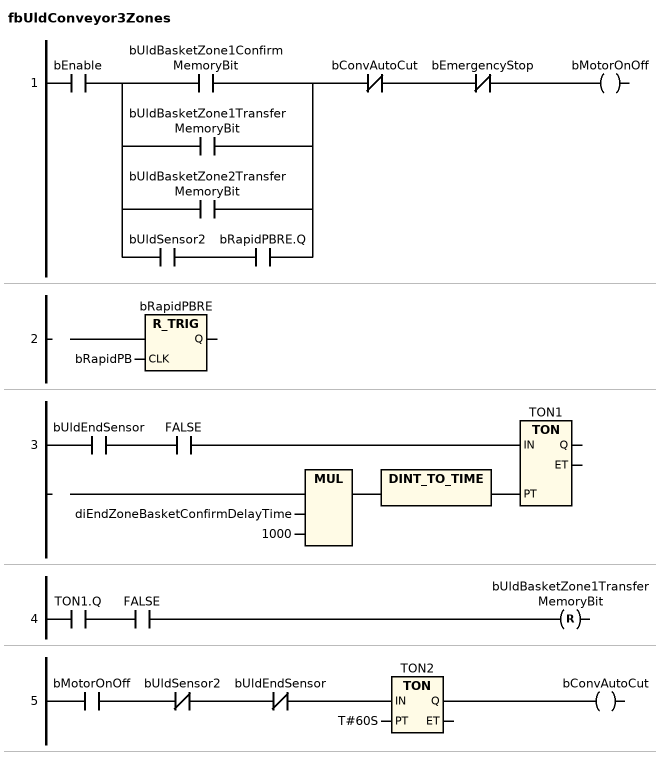
// NETWORK 1
bMotorOnOff := (bEnable AND (bUldBasketZone1ConfirmMemoryBit OR bUldBasketZone1TransferMemoryBit OR bUldBasketZone2TransferMemoryBit OR bUldSensor2 AND bRapidPBRE.Q)) AND NOT bConvAutoCut AND NOT bEmergencyStop;

// NETWORK 2
bRapidPBRE(CLK := bRapidPB); // R_TRIG

// NETWORK 3
TON1(IN := bUldEndSensor AND FALSE, PT := DINT_TO_TIME(diEndZoneBasketConfirmDelayTime * 1000)); // TON

// NETWORK 4
bUldBasketZone1TransferMemoryBit R= TON1.Q AND FALSE;

// NETWORK 5
TON2(IN := bMotorOnOff AND NOT bUldSensor2 AND NOT bUldEndSensor, PT := T#60S); // TON
bConvAutoCut := TON2.Q;

END_FUNCTION_BLOCK

// ---- FBs/B_JKS_CustomFB/Other/fb_ArmBasketRotateCtrl.TcPOU
FUNCTION_BLOCK fb_ArmBasketRotateCtrl
VAR_INPUT
	bEn 							: BOOL;
	bStart			 			: BOOL;
	bRotateBasketRS_Cw			: BOOL;
	bRotateBasketRS_Ccw		: BOOL;
	bRotateBasketRS_Lock		: BOOL;
	bRotateBasketRS_Unlock		: BOOL;
	bDeactivatedMode 			: BOOL;
	iRotateBasketDelayTimeSV	: INT;
END_VAR
VAR_OUTPUT
	bRotateBasketAV_Cw			: BOOL;
	bRotateBasketAV_Ccw		: BOOL;
	bRotateBasketAV_Lock		: BOOL;
	bRotateBasketAV_Unlock		: BOOL;

END_VAR
VAR

	bStep1: BOOL;
	bStep2: BOOL;
	tRotateBasketDelay: TON;
END_VAR

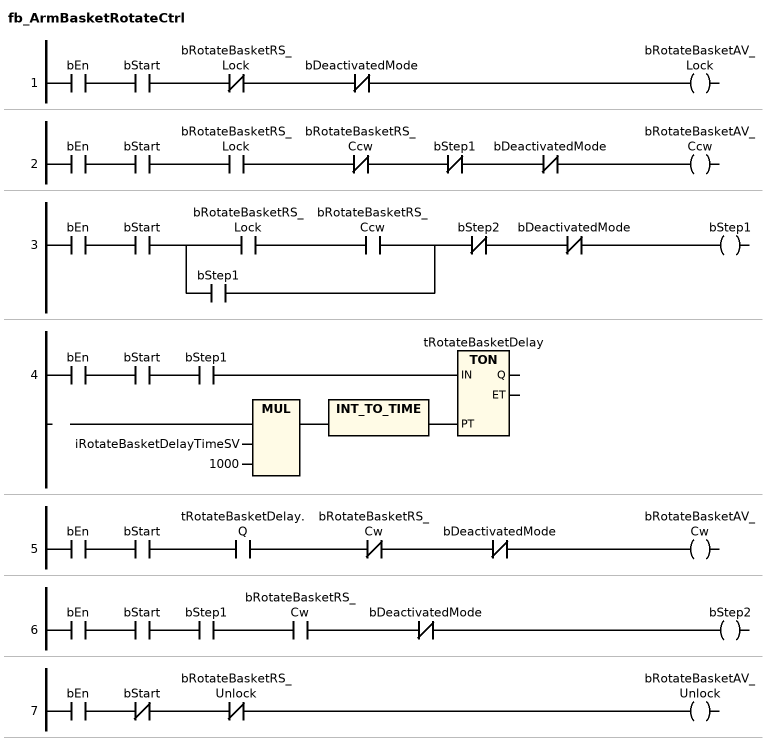
// NETWORK 1
bRotateBasketAV_Lock := bEn AND bStart AND NOT bRotateBasketRS_Lock AND NOT bDeactivatedMode;

// NETWORK 2
bRotateBasketAV_Ccw := bEn AND bStart AND bRotateBasketRS_Lock AND NOT bRotateBasketRS_Ccw AND NOT bStep1 AND NOT bDeactivatedMode;

// NETWORK 3
bStep1 := (bEn AND bStart AND (bRotateBasketRS_Lock AND bRotateBasketRS_Ccw OR bStep1)) AND NOT bStep2 AND NOT bDeactivatedMode;

// NETWORK 4
tRotateBasketDelay(IN := bEn AND bStart AND bStep1, PT := INT_TO_TIME(iRotateBasketDelayTimeSV * 1000)); // TON

// NETWORK 5
bRotateBasketAV_Cw := bEn AND bStart AND tRotateBasketDelay.Q AND NOT bRotateBasketRS_Cw AND NOT bDeactivatedMode;

// NETWORK 6
bStep2 := bEn AND bStart AND bStep1 AND bRotateBasketRS_Cw AND NOT bDeactivatedMode;

// NETWORK 7
bRotateBasketAV_Unlock := bEn AND NOT bStart AND NOT bRotateBasketRS_Unlock;

END_FUNCTION_BLOCK

// ---- FBs/B_JKS_CustomFB/Other/fb_StnCylinderInOutCtrl.TcPOU
FUNCTION_BLOCK fb_StnCylinderInOutCtrl
VAR_INPUT
	bEn 								: BOOL;
	bStart			 				: BOOL;
	bCylinderBasketRS_Front			: BOOL;
	bCylinderBasketRS_Back			: BOOL;
	bDeactivatedMode 				: BOOL;
	iCylinderBasketBackDelayTimeSV	: INT;
	iCylinderBasketFrontDelayTimeSV	: INT;

END_VAR
VAR_OUTPUT
	bCylinderBasketAV_Front		: BOOL;
	bCylinderBasketAV_Back		: BOOL;

END_VAR
VAR

	bStep1: BOOL;
	bStep2: BOOL;
	tCylinderBasketBackDelay: TON;
	tCylinderBasketFrontDelay: TON;
END_VAR

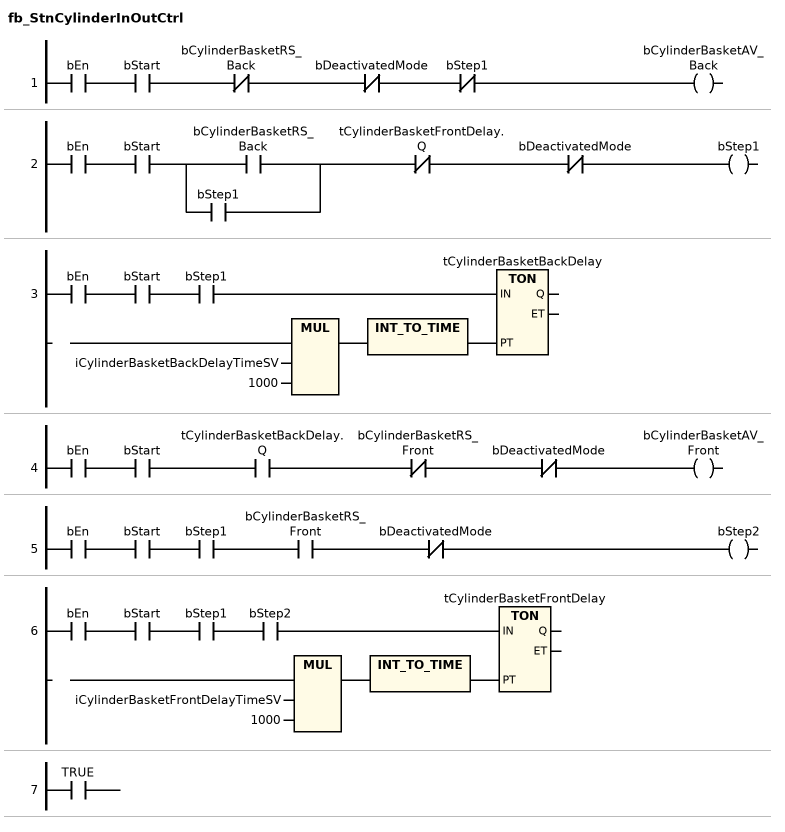
// NETWORK 1
bCylinderBasketAV_Back := bEn AND bStart AND NOT bCylinderBasketRS_Back AND NOT bDeactivatedMode AND NOT bStep1;

// NETWORK 2
bStep1 := (bEn AND bStart AND (bCylinderBasketRS_Back OR bStep1)) AND NOT tCylinderBasketFrontDelay.Q AND NOT bDeactivatedMode;

// NETWORK 3
tCylinderBasketBackDelay(IN := bEn AND bStart AND bStep1, PT := INT_TO_TIME(iCylinderBasketBackDelayTimeSV * 1000)); // TON

// NETWORK 4
bCylinderBasketAV_Front := bEn AND bStart AND tCylinderBasketBackDelay.Q AND NOT bCylinderBasketRS_Front AND NOT bDeactivatedMode;

// NETWORK 5
bStep2 := bEn AND bStart AND bStep1 AND bCylinderBasketRS_Front AND NOT bDeactivatedMode;

// NETWORK 6
tCylinderBasketFrontDelay(IN := bEn AND bStart AND bStep1 AND bStep2, PT := INT_TO_TIME(iCylinderBasketFrontDelayTimeSV * 1000)); // TON

// NETWORK 7

END_FUNCTION_BLOCK

// ---- FBs/B_JKS_CustomFB/Other/ReservoirTankDrain.TcPOU
FUNCTION_BLOCK ReservoirTankDrain
VAR_INPUT

	bMainOnOff:BOOL;
	iDrainCollectTimer:INT;
	iDrainTransferTimer:INT;
	iDrainingTimer:INT;
	bDirectDrainST:BOOL;
END_VAR

VAR_OUTPUT

	bReservoirDrainAv1:BOOL;
	bReservoirDrainAv2:BOOL;
	ProcessComplete:BOOL;
END_VAR

VAR
	Timer1: DOWN_COUNT_TIMER;
	CollectTimerComplete: BOOL;
	Timer2: DOWN_COUNT_TIMER;
	TransferComplete: BOOL;
	Timer3: DOWN_COUNT_TIMER;
	DrainComplete: BOOL;
	DelayComplete: TON;
	iDrainCollectCounDown: INT;
	iDrainTransferCountDown: INT;
	iDrainCountDown: INT;
	bDirectDrainInProcess: BOOL;
END_VAR

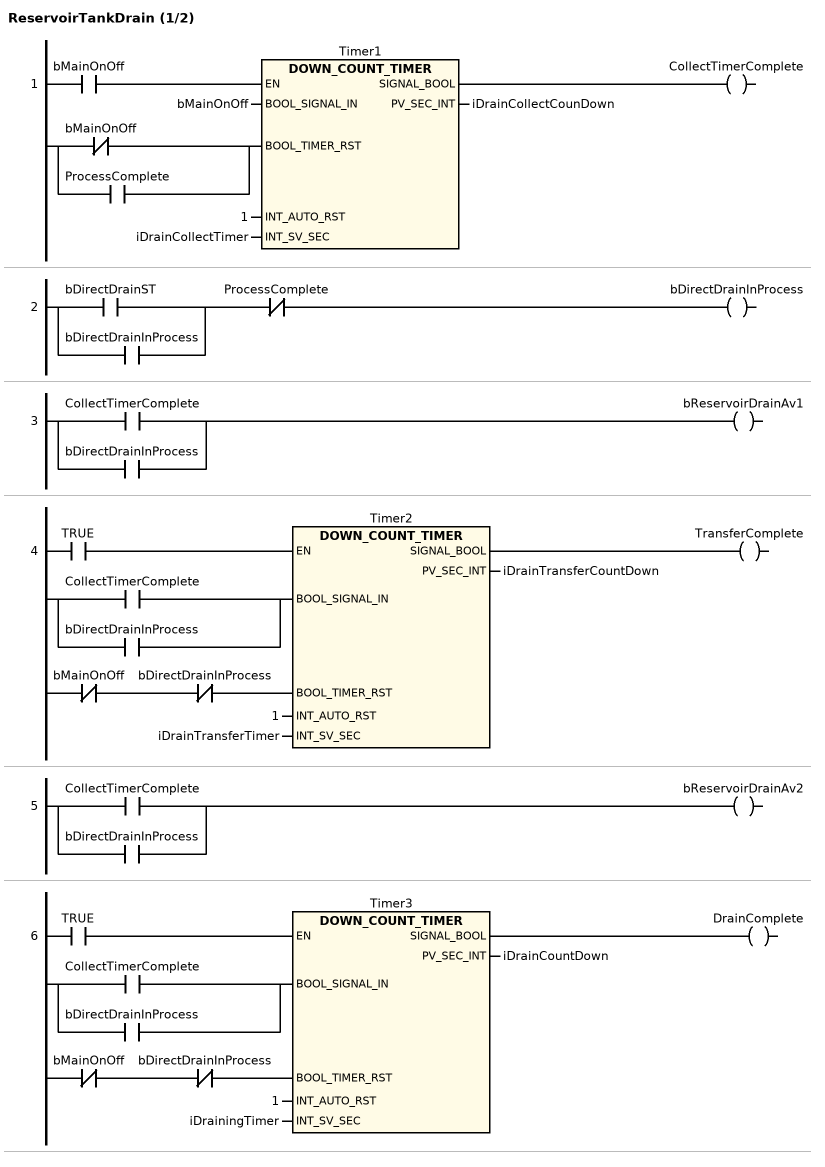
// NETWORK 1
IF bMainOnOff THEN
    Timer1(
        BOOL_SIGNAL_IN := bMainOnOff,
        BOOL_TIMER_RST := NOT bMainOnOff OR ProcessComplete,
        INT_AUTO_RST := 1,
        INT_SV_SEC := iDrainCollectTimer,
        PV_SEC_INT => iDrainCollectCounDown); // DOWN_COUNT_TIMER
END_IF
CollectTimerComplete := Timer1.SIGNAL_BOOL;

// NETWORK 2
bDirectDrainInProcess := (bDirectDrainST OR bDirectDrainInProcess) AND NOT ProcessComplete;

// NETWORK 3
bReservoirDrainAv1 := CollectTimerComplete OR bDirectDrainInProcess;

// NETWORK 4
Timer2(
    BOOL_SIGNAL_IN := CollectTimerComplete OR bDirectDrainInProcess,
    BOOL_TIMER_RST := NOT bMainOnOff AND NOT bDirectDrainInProcess,
    INT_AUTO_RST := 1,
    INT_SV_SEC := iDrainTransferTimer,
    PV_SEC_INT => iDrainTransferCountDown); // DOWN_COUNT_TIMER
TransferComplete := Timer2.SIGNAL_BOOL;

// NETWORK 5
bReservoirDrainAv2 := CollectTimerComplete OR bDirectDrainInProcess;

// NETWORK 6
Timer3(
    BOOL_SIGNAL_IN := CollectTimerComplete OR bDirectDrainInProcess,
    BOOL_TIMER_RST := NOT bMainOnOff AND NOT bDirectDrainInProcess,
    INT_AUTO_RST := 1,
    INT_SV_SEC := iDrainingTimer,
    PV_SEC_INT => iDrainCountDown); // DOWN_COUNT_TIMER
DrainComplete := Timer3.SIGNAL_BOOL;

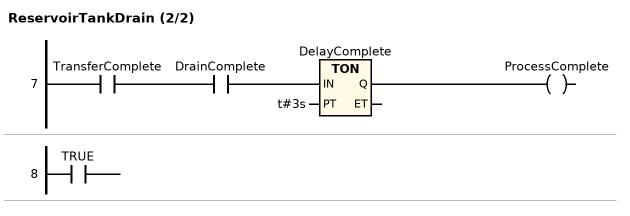
// NETWORK 7
DelayComplete(IN := TransferComplete AND DrainComplete, PT := t#3s); // TON
ProcessComplete := DelayComplete.Q;

// NETWORK 8

END_FUNCTION_BLOCK

// ---- FBs/B_JKS_OldFB/Timer/DOWN_COUNT_TIMER.TcPOU
FUNCTION_BLOCK DOWN_COUNT_TIMER
VAR_INPUT
	BOOL_SIGNAL_IN: BOOL;
	BOOL_TIMER_RST: BOOL;
	INT_AUTO_RST: INT;
	INT_SV_SEC: INT;
END_VAR
VAR_OUTPUT
	SIGNAL_BOOL: BOOL;
	PV_SEC_INT: INT;
END_VAR
VAR
	DF_1: R_TRIG;
	DF_2: R_TRIG;
	M1: BOOL;
	M2: BOOL;

	T100: TON;
	T101: TON;
	M100: BOOL;
	M101: BOOL;
	M200: BOOL;

	M110: BOOL;
	M300: BOOL;
END_VAR
VAR // added by the converter: edge detectors and wires of the graphical bodies
    _w1, _w2 : INT;
END_VAR

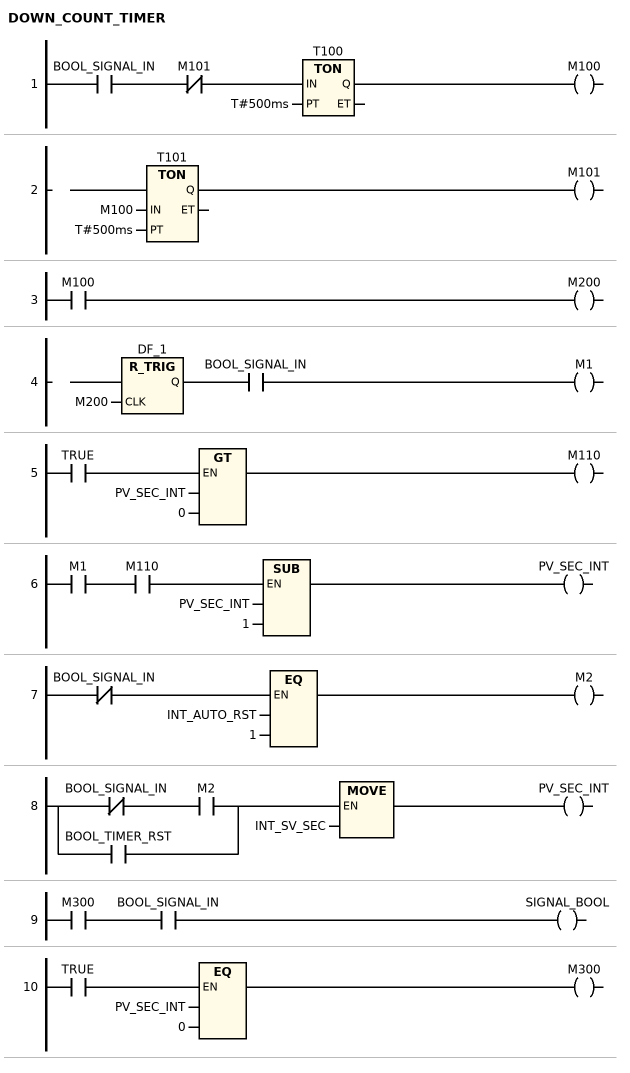
// NETWORK 1
T100(IN := BOOL_SIGNAL_IN AND NOT M101, PT := T#500ms); // TON
M100 := T100.Q;

// NETWORK 2
T101(IN := M100, PT := T#500ms); // TON
M101 := T101.Q;

// NETWORK 3
M200 := M100;

// NETWORK 4
DF_1(CLK := M200); // R_TRIG
M1 := DF_1.Q AND BOOL_SIGNAL_IN;

// NETWORK 5
M110 := PV_SEC_INT > 0;

// NETWORK 6
IF M1 AND M110 THEN _w1 := PV_SEC_INT - 1; END_IF
PV_SEC_INT := _w1;

// NETWORK 7
M2 := NOT BOOL_SIGNAL_IN AND INT_AUTO_RST = 1;

// NETWORK 8
IF NOT BOOL_SIGNAL_IN AND M2 OR BOOL_TIMER_RST THEN _w2 := INT_SV_SEC; END_IF
PV_SEC_INT := _w2;

// NETWORK 9
SIGNAL_BOOL := M300 AND BOOL_SIGNAL_IN;

// NETWORK 10
M300 := PV_SEC_INT = 0;

END_FUNCTION_BLOCK

// ---- FBs/B_JKS_CustomFB/Other/ReservoirTankDrainNIL.TcPOU
FUNCTION_BLOCK ReservoirTankDrainNIL
VAR_INPUT

	bMainOnOff:BOOL;
	iDrainCollectTimer:INT;
	iDrainTransferTimer:INT;
	iDrainingTimer:INT;
	bDirectDrainST:BOOL;
END_VAR

VAR_OUTPUT

	bReservoirDrainAv1:BOOL;
	bReservoirDrainAv2:BOOL;
	ProcessComplete:BOOL;
END_VAR

VAR
	Timer1: DOWN_COUNT_TIMER;
	CollectTimerComplete: BOOL;
	Timer2: DOWN_COUNT_TIMER;
	TransferComplete: BOOL;
	Timer3: DOWN_COUNT_TIMER;
	DrainComplete: BOOL;
	DelayComplete: TON;
	Coundown: INT;
	bDirectDrainInProcess: BOOL;
END_VAR

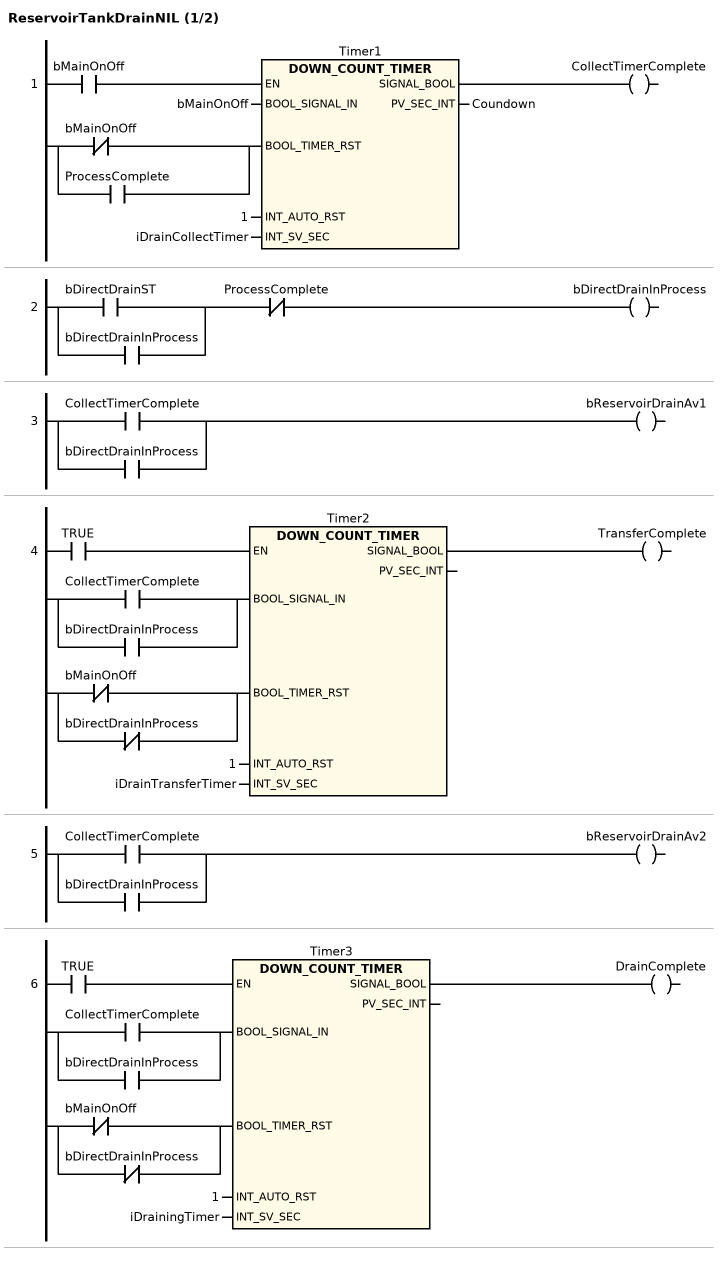
// NETWORK 1
IF bMainOnOff THEN
    Timer1(
        BOOL_SIGNAL_IN := bMainOnOff,
        BOOL_TIMER_RST := NOT bMainOnOff OR ProcessComplete,
        INT_AUTO_RST := 1,
        INT_SV_SEC := iDrainCollectTimer,
        PV_SEC_INT => Coundown); // DOWN_COUNT_TIMER
END_IF
CollectTimerComplete := Timer1.SIGNAL_BOOL;

// NETWORK 2
bDirectDrainInProcess := (bDirectDrainST OR bDirectDrainInProcess) AND NOT ProcessComplete;

// NETWORK 3
bReservoirDrainAv1 := CollectTimerComplete OR bDirectDrainInProcess;

// NETWORK 4
Timer2(
    BOOL_SIGNAL_IN := CollectTimerComplete OR bDirectDrainInProcess,
    BOOL_TIMER_RST := NOT bMainOnOff OR NOT bDirectDrainInProcess,
    INT_AUTO_RST := 1,
    INT_SV_SEC := iDrainTransferTimer); // DOWN_COUNT_TIMER
TransferComplete := Timer2.SIGNAL_BOOL;

// NETWORK 5
bReservoirDrainAv2 := CollectTimerComplete OR bDirectDrainInProcess;

